(* CODESYS project Function Blocks.export

Project tree, tasks and I/O mapping:
  Function Blocks/
    Actuator/
      function block Actuator [ST]: Close, Open
      function block ActuatotLockAssermbler [ST]: AssembleClosingLockCameraClosed, AssembleClosingLockCameraOpen, AssembleOpenAndUpLock, AssembleOpenvacuumLocked
    DepositeProccess/
      function block absCommonDepositeProcessUnitExplorer [ST]: AddDepositeDevice, AddMaterialRawRateData, AddMaterialShutter, AddQuartzReset, AddQuartzShutter, AddThinknessData, DepositeDeviceCheck, DepositeDeviceStart, DepositeDeviceStop, GetDepositeDevice, GetDepositeDeviceSetting, GetMaterialRawRateData, GetMatertialShutter, GetQuartzReset, GetQuartzShutter, GetThinknessData, InitSelectedPosition, MaterialShutterClose, MaterialShutterOpen, NullPtrCheck, QuartzShutterClose, QuartzShutterOpen, QuartzThinknessReset, _getManipulatingVariable, ActualRawRate, ActualThinkness, DeviceManipulatingVariable, DevicePosition, isMaterialShutterAutoMode, isMaterialShutterRemoteMode, SelectedDevice, SelectedDeviceManipualtedValueFB, SelectedDeviceManipulatingValue, SelectedDeviceSetting
      function block absDepositeUnit [ST]: AddDepositeDevice, AddMaterialShutter, AddQuartzResetCommand, AddQuartzShutter, AddRawRateData, AddThinknessData, CloseMaterialShutter, CloseQuartzShutter, OpenMaterialShutter, OpenQuartzShutter, ResetThinkness, StartDepositeDevice, StopDepositeDevice, DeviceAutoMode, DeviceManipulatingVariable, MaterialShutterAutoMode, MaxManipulatingVariable, MinManipulatingVariable, RawRate, Thinkness
      function block CommonDepositeProcess [ST]: getPreheatTimerTrigger, ProcessStage, _acknowledgment, _calcSP, _error, _getSelectedDevice, _initData, _limitSpeedDeposite, _pidAutoMode, _pidManualMode, _predepositeHeating, _qartzOpen, _qartzSensoreHeating, _quartzOpenedDelay, _resultHandler, _sourceShutterOpen, _startHeater, _startPreheatTimer, _startQuartzHeatingTimer, _startQuartzOpenDelayTimer, _stopDeposite, _stopPreheatTimer, _stopQuartzHeatingTimer, _stopQuartzOpenDelayTimer, _TimerCall, _waitCommand, DepositeSPFromPID, depositeThinknessLimit, Dkoeff, getPreheatLeftTimeSecond, getPreheatTime, getQuartzHeatingLeftTimeSecond, getQuartzHeatingTime, getQuartzOpenDelayLeftTimeSecond, getQuartzOpenDelayTime, Ikoeff, PIDAutoMode, pidAutoModeSP, PIDManualVariable, PIDYMax, PIDYMin, Pkoeff, RawRate, SelectedDevicePosition, _preheatTimerComplete, _quartzHeatingTimerComplete, _quartzOpenDelayTimerComplete
      function block fbDepositeProccess [ST]: AssemblePermition, CalcSP, InitTimers, SelectDepositeSource, Update, getPreheatTimeLeftSecond, setGorn1, setGorn2, setGorn3, setGornSetting1, setGornSetting2, setGornSetting3, setQartzReset1, setQartzReset2, setQartzReset3, setQuartzShutter1, setQuartzShutter2, setQuartzShutter3, setRawRate1, setRawRate2, setRawRate3, setShutter1, setShutter2, setShutter3, setShutterSetting1, setShutterSetting2, setShutterSetting3, setThinkness1, setThinkness2, setThinkness3
      function block fbGornDepositeProccess [ST]: AssemblePermition, CalcSP, InitTimers, SelectDepositeSource, Update, getPreheatTimeLeftSecond, setGorn1, setGorn2, setGorn3, setGornSetting1, setGornSetting2, setGornSetting3, setQartzReset1, setQartzReset2, setQartzReset3, setQuartzShutter1, setQuartzShutter2, setQuartzShutter3, setRawRate1, setRawRate2, setRawRate3, setShutter1, setShutter2, setShutter3, setShutterSetting1, setShutterSetting2, setShutterSetting3, setThinkness1, setThinkness2, setThinkness3
      function block GornDepositeUnit [ST]: _addDepositeDevice, _deviceAutoMode, _deviceManipulatingVariableGet, _deviceManipulatingVariableSet, _maxManipulatingVariable, _minManipulatingVariable, _startDepositeDevice, _stopDepositeDevice
      function block HeaterDepositeUnit [ST]: _addDepositeDevice, _deviceAutoMode, _deviceManipulatingVariableGet, _deviceManipulatingVariableSet, _maxManipulatingVariable, _minManipulatingVariable, _startDepositeDevice, _stopDepositeDevice
    Driver/
      function block fbBSDDriver [ST]
    GasRegulator/
      function block fbGasRegulator [ST]: CalcRRGSPwithCoeff
    GeneralBuffer/
      function block fbGeneralBuffer [ST]: AddElement, AddStruct, ClearBuffer, getBufferAddres, getBufferLength
    Gorn/
      function block Gorn [ST]
    Heater/
      data type udtHeater
      data type udtHeaterSetting
      function block fbHeater [ST]
    Inficon/
      function block fbInficon [ST]: ADD_Sensore, CalcCRC, GetMateriaFiltredRate, HCPub, HelloCommand, RemoteGeneralAction, SensoreStatus
      function block fbInficonQuery [ST]: General, Material, ProcessMaterial, Sensor, Source
      function block fbInficonRemote [ST]: General, MaterialAction
      function block fbInficonStatus [ST]: Material, Sensor
      function block fbInficonUpdate [ST]: General, Material, ProcessMaterial, Sensor, Source
    IPS/
      function block IPSIon [ST]
      function block IPSIonModbus [ST]
    Pumps/
      Interlock/
        function block PumpsInterlock [ST]: AssembleFVPInterlock, AssembleFVPOpenCameraLocked, AssembleTMPFVPTurnOffLocked, AssembleTMPInterlock, AssembleTMPPressureLocked
      function block FVP [ST]: AssebleLock
      function block TMP [ST]: AssembleLock, AssembleLockWithSHV, RotateSignalAssemble, StatusAssemble, StatusTimerLogic
      function block TMPPfifer [ST]
    RRG/
      function block fbRRG [ST]
      function block fbRRGModbus [ST]: AssembleStatusFromFieldStatus2, ConvertModbusSPFeedbackToSPfeedback, ConvertModbusValueFbTovalueFb, ConvertValueSPtoModbusData, UnmarshalModbusFlagStatus1ToRRGFeedback
    Shutter/
      function block fbShutter [ST]
    TRM-151/
      Middleware/
        function block MC_ChannelView_ChannelTRM [ST]
        function block MC_InputView_InputTRM [ST]
        function block MC_OperatingView_OperatingTRM [ST]
        function block MC_OutputView_OutputTRM [ST]
        function block MC_ProgramOfTecholog_ProgramOfTechnologTRM [ST]
        function block MC_RegulatorView_RegulatorTRM [ST]
      Pooling/
        function block MC_TRMPooling [ST]
    TRM_View/
      function block MC_Heater [ST]
      function block MC_TRMChannel [ST]
      function block MC_TRMInput [ST]
      function block MC_TRMOperating [ST]
      function block MC_TRMOutput [ST]
      function block MC_TRMProgramOfTechnolog [ST]
      function block MC_TRMRegulator [ST]
    VacuumCamera/
      Pumping/
        function block VacuumCameraWithoutSHV [ST]: StartDevacuumProcessCommand, StartVacuumProcessCommand, StopVacuumProcessCommand, CancelOperatorCommand, CheckFVPSelect, CheckingFVP, CloseAllvalves, devcuumProcessOpenCam, ErrorHandle, forvacuumingProcess, forvacuumingWithTMPValve, OperatorCommandHandler, operatorStopAnyProcess, startDevacuumProcess, startTMP, startVacuumProcess, stopFVP, stopTMP, stopVacuumProcess, waitVacuumingProcess, isAllValvesClosed, isFVPChecked, isOperatorCommandEntryLocked, isVacuumCameraClosed, isVacuumCameraDeviceAutoMode
        function block VacuumingCameraWithSHV [ST]: CloseAllValves, Devacuum, Revacuum, StartUnit, StopUnit, ValveOpen, _commandHandler, _commandRouter, _resetAllCommand, _resetProcess, isAllvalveClosed
      global variables VacuumCameraErrorsList
      global variables VacuumCameraStatusList
    VacuumSensore/
      ConverExp/
        function ConverPressureToHmi [ST]
        function LessPressure [ST]
        function More [ST]
      function block VacuumSensore [ST]: CalcPressure
    Valves/
      global variables ValveInterlockStatus
      function block Valve [ST]
      function block ValvesInterlock [ST]: AnotherValveOpenInterlock, AssembleSHVLockStatus, AssembleValveStatus, LowPressureInterlock
    function block DiscreteInput [ST]
    function block DiscreteOutput [ST]
    function block HeatFloatSensore [ST]: isFloatL, isFloatLL, isTemepratureHH, isTemperatureH
    function block OwenAnalogInput [ST]
    function block TMPBreakingValve [ST]
*)

// Function Blocks/Heater/udtHeater
TYPE udtHeater :
STRUCT
	xPowerOn:		BOOL;
	xError:			BOOL;
	xLock:			BOOL;
	xManualCommand:	BOOL;
	xAutoCommand:	BOOL;
	xReset:			BOOL;
	xCommand: 		BOOL;
	Temepature:		REAL;
	rPower:			REAL;
	wState:			BYTE;
END_STRUCT
END_TYPE

// Function Blocks/Heater/udtHeaterSetting
TYPE udtHeaterSetting :
STRUCT
	rMinPower:		REAL:=0;
	rMaxPower:		REAL:=100.0;
	rManualPower: 	REAL;
	rAutoPower:		REAL;
	rSetpointTemperature: REAL;
	P: REAL:=2.0;
	I:REAL:=15.0;
	D:REAL:=0.0;
	rMinimalAccessPressure:	REAL:=0.003;
	xAutoMode:		BOOL;
	xServiceMode:	BOOL;
	xManualPower: BOOL;
	
END_STRUCT
END_TYPE

// Function Blocks/VacuumCamera/VacuumCameraErrorsList
{attribute 'qualified_only'}
VAR_GLOBAL CONSTANT
	NO_ERROR: 						WORD:=16#00;
	ALL_DEVICES_DONT_HAVE_AUTOMODE: WORD:=16#02;
	VACUUM_CAMERA_OPEN: 			WORD:=16#03;
	FVP_CHECK_FAIL:					WORD:=16#04;
	TMP_ERROR_FROM_START:			WORD:=16#05;
END_VAR

// Function Blocks/VacuumCamera/VacuumCameraStatusList
{attribute 'qualified_only'}
VAR_GLOBAL CONSTANT
	SYSTEM_READY_AND_WAIT_COMMAND: 			WORD:=00;
	SYSTEM_HAS_ERROR:						WORD:=01;
	STOP_ANY_PROCESS_SIGNAL_FROM_OPERATOR:	WORD:=02;
	START_VACUUM_PROCESS:					WORD:=03;
	CHECK_FVP_START_FVP:					WORD:=04;
	CHECK_FVP_START_TIMER:					WORD:=05;
	CHECK_FVP_COMPLETE:						WORD:=06;
	CHECK_FVP_FAILED:						WORD:=07;
	START_FORVAC_PROCESS:					WORD:=08;
	FORVAC_COMPLETE:						WORD:=09;	
	FORVAC_WITH_TMP_VALVE:					WORD:=10;
	FORVAC_WITH_TMP_VALVE_COMPLETE:			WORD:=11;
	TMP_IS_STARTED:							WORD:=12;
	TMP_IS_RUN:								WORD:=13;
	CAMERA_IS_VACUUMING:					WORD:=14;
	VACUUM_DONE:							WORD:=15;
	STOP_TMP_PROCESS:						WORD:=16;
	STOP_FVP_PROCESS:						WORD:=17;
	STOP_TMP_OPEN_BAV3:						WORD:=18;
	STOP_TMP_DONE:							WORD:=19;
	STOP_FVP_PROCESS_DONE:					WORD:=20;
	STOP_SYSTEM_COMPLITE:					WORD:=21;
	OPERATOR_STOPED_PROCESS_COMPLETE:		WORD:=22;
	BAV3OPENED:								WORD:=23;
	FVP_CHECK_COMPLETED:					WORD:=24;
END_VAR

// Function Blocks/Valves/ValveInterlockStatus
{attribute 'qualified_only'}
VAR_GLOBAL CONSTANT
	NO_LOCK: WORD:=0;//Нет блокировок
	LOW_PRESSURE_INTERLOCK: WORD:=1;//Блокирвока из-за недостаточного давления в пневмосистеме
	LOCKER_VALVE_OPENED: WORD:=2;//Блокировка из-за открытия блокирующего клапана
	HIGH_PRESSURE_INTERLOCK: WORD:=3;// Высокое давление в линии
END_VAR

// Function Blocks/DepositeProccess/absCommonDepositeProcessUnitExplorer/_addDepositeDevice
METHOD PROTECTED ABSTRACT _addDepositeDevice : dpResult
VAR_INPUT
	iPosition: INT;
	ptrDepositeDevice: POINTER TO BYTE;
	ptrDepositeDeviceSetting: POINTER TO BYTE;
END_VAR

// Function Blocks/DepositeProccess/absCommonDepositeProcessUnitExplorer/_addMaterialRawRateData
METHOD PROTECTED ABSTRACT _addMaterialRawRateData : dpResult
VAR_INPUT
	ptrMaterialRawRateData	: POINTER TO BYTE;
	iPosition	: INT;
END_VAR

// Function Blocks/DepositeProccess/absCommonDepositeProcessUnitExplorer/_addMaterialShutter
METHOD PROTECTED ABSTRACT _addMaterialShutter : dpResult
VAR_INPUT
	ptrMaterialShutter	: POINTER TO BYTE;
	ptrMaterialShutterSetting	: POINTER TO BYTE;
	iPosition	: INT;
END_VAR

// Function Blocks/DepositeProccess/absCommonDepositeProcessUnitExplorer/_addQuartzReset
METHOD PROTECTED ABSTRACT _addQuartzReset : dpResult
VAR_INPUT
	ptrQuartzReset	: POINTER TO BYTE;
	iPosition	: INT;
END_VAR

// Function Blocks/DepositeProccess/absCommonDepositeProcessUnitExplorer/_addQuartzShutter
METHOD PROTECTED ABSTRACT _addQuartzShutter : dpResult
VAR_INPUT
	ptrQuartzShutter	: POINTER TO udtDiscreteSignal;
	iPosition	: INT;
END_VAR

// Function Blocks/DepositeProccess/absCommonDepositeProcessUnitExplorer/_addThinknessData
METHOD PROTECTED ABSTRACT _addThinknessData : dpResult
VAR_INPUT
	ptrThinknessData	: POINTER TO REAL;
	iPosition	: INT;
END_VAR

// Function Blocks/DepositeProccess/absCommonDepositeProcessUnitExplorer/_depositeDeviceCheck
METHOD PROTECTED ABSTRACT _depositeDeviceCheck : dpResult
VAR_INPUT
	Status: REFERENCE TO dpuStatus;
END_VAR

// Function Blocks/DepositeProccess/absCommonDepositeProcessUnitExplorer/_depositeDeviceStart
METHOD PROTECTED ABSTRACT _depositeDeviceStart : dpResult
VAR_INPUT
END_VAR

// Function Blocks/DepositeProccess/absCommonDepositeProcessUnitExplorer/_depositeDeviceStop
METHOD PROTECTED ABSTRACT _depositeDeviceStop : dpResult
VAR_INPUT
END_VAR

// Function Blocks/DepositeProccess/absCommonDepositeProcessUnitExplorer/_getDepositeDevice
METHOD PROTECTED ABSTRACT _getDepositeDevice : POINTER TO BYTE
VAR_INPUT
	iPostion	: INT;
END_VAR
VAR_OUTPUT
	Result	: dpResult;
END_VAR

// Function Blocks/DepositeProccess/absCommonDepositeProcessUnitExplorer/_getDepositeDeviceSetting
METHOD PROTECTED ABSTRACT _getDepositeDeviceSetting : POINTER TO BYTE
VAR_INPUT
	iPosition	: INT;
END_VAR
VAR_OUTPUT
	Result	: dpResult;
END_VAR

// Function Blocks/DepositeProccess/absCommonDepositeProcessUnitExplorer/_getMaterialRawRateData
METHOD PROTECTED ABSTRACT _getMaterialRawRateData : POINTER TO REAL
VAR_INPUT
	iPosition	: INT;
END_VAR
VAR_OUTPUT
	Result	: dpResult;
END_VAR

// Function Blocks/DepositeProccess/absCommonDepositeProcessUnitExplorer/_getMaterialShutter
METHOD PROTECTED ABSTRACT _getMaterialShutter : POINTER TO udtShutter
VAR_INPUT
	iPosition	: INT;
END_VAR
VAR_OUTPUT
	Result	: dpResult;
END_VAR

// Function Blocks/DepositeProccess/absCommonDepositeProcessUnitExplorer/_getMaterialShutterSetting
METHOD PROTECTED ABSTRACT _getMaterialShutterSetting : POINTER TO udtShutterSetting
VAR_INPUT
	iPosition	: INT;
END_VAR
VAR_OUTPUT
	Result	: dpResult;
END_VAR

// Function Blocks/DepositeProccess/absCommonDepositeProcessUnitExplorer/_getQuartzReset
METHOD PROTECTED ABSTRACT _getQuartzReset : POINTER TO BOOL
VAR_INPUT
	iPosition	: INT;
END_VAR
VAR_OUTPUT
	Result	: dpResult;
END_VAR

// Function Blocks/DepositeProccess/absCommonDepositeProcessUnitExplorer/_getQuartzShutter
METHOD PROTECTED ABSTRACT _getQuartzShutter : POINTER TO udtDiscreteSignal
VAR_INPUT
	iPosition	: INT;
END_VAR
VAR_OUTPUT
	Result	: dpResult;
END_VAR

// Function Blocks/DepositeProccess/absCommonDepositeProcessUnitExplorer/_getSelectedDepositeDevice
METHOD PROTECTED ABSTRACT _getSelectedDepositeDevice : POINTER TO BYTE
VAR_INPUT
END_VAR

// Function Blocks/DepositeProccess/absCommonDepositeProcessUnitExplorer/_getSelectedDeviceManipulatingValue
{warning 'Проследить за всеми использованиями данного метода'}
METHOD PROTECTED ABSTRACT _getSelectedDeviceManipulatingValue : POINTER TO BYTE
VAR_INPUT
END_VAR

// Function Blocks/DepositeProccess/absCommonDepositeProcessUnitExplorer/_getSelectedDeviceManipulatingValueFB
{warning 'Проследить за всеми использованиями данного метода'}
METHOD PROTECTED ABSTRACT _getSelectedDeviceManipulatingValueFB : POINTER TO BYTE
VAR_INPUT
END_VAR

// Function Blocks/DepositeProccess/absCommonDepositeProcessUnitExplorer/_getSelectedDeviceSetting
METHOD PROTECTED ABSTRACT _getSelectedDeviceSetting : POINTER TO BYTE
VAR_INPUT
END_VAR

// Function Blocks/DepositeProccess/absCommonDepositeProcessUnitExplorer/_getThinknessData
METHOD PROTECTED ABSTRACT _getThinknessData : POINTER TO REAL
VAR_INPUT
	iPosition	: INT;
END_VAR
VAR_OUTPUT
	Result	: dpResult;
END_VAR

// Function Blocks/DepositeProccess/absCommonDepositeProcessUnitExplorer/_initSelectedPosition
//инициализация выбранной позиции. Устройства нагрева
METHOD PROTECTED ABSTRACT _initSelectedPosition : dpResult
VAR_INPUT
	iPosition	: INT;
END_VAR
VAR_OUTPUT
	Status	: dpuStatus;
END_VAR

// Function Blocks/DepositeProccess/absCommonDepositeProcessUnitExplorer/_isDepositeDeviceAutoMode
METHOD PROTECTED ABSTRACT _isDepositeDeviceAutoMode : dpResult
VAR_INPUT
END_VAR

// Function Blocks/DepositeProccess/absCommonDepositeProcessUnitExplorer/_isDepositeDeviceBlocked
METHOD PROTECTED ABSTRACT _isDepositeDeviceBlocked : dpResult
VAR_INPUT
END_VAR

// Function Blocks/DepositeProccess/absCommonDepositeProcessUnitExplorer/_isDepositeDeviceModbusConnected
METHOD PROTECTED ABSTRACT _isDepositeDeviceModbusConnected : dpResult
VAR_INPUT
END_VAR

// Function Blocks/DepositeProccess/absCommonDepositeProcessUnitExplorer/_materialShutterClose
METHOD PROTECTED ABSTRACT _materialShutterClose : dpResult
VAR_INPUT
END_VAR

// Function Blocks/DepositeProccess/absCommonDepositeProcessUnitExplorer/_nullPtrCheck
METHOD PROTECTED ABSTRACT _nullPtrCheck : dpResult
VAR_INPUT
END_VAR

// Function Blocks/DepositeProccess/absCommonDepositeProcessUnitExplorer/_setManipulatingVariable
METHOD PROTECTED ABSTRACT _setManipulatingVariable : dpResult
VAR_INPUT
	Value:REAL;
END_VAR

// Function Blocks/DepositeProccess/absDepositeUnit/_addDepositeDevice
METHOD  ABSTRACT _addDepositeDevice : dpResult
VAR_INPUT
	ptrDevice	: 			POINTER TO BYTE;
	ptrDeviceSetting	: 	POINTER TO BYTE;
END_VAR

// Function Blocks/DepositeProccess/absDepositeUnit/_deviceAutoMode
METHOD PROTECTED ABSTRACT _deviceAutoMode : BOOL
VAR_INPUT
END_VAR

// Function Blocks/DepositeProccess/absDepositeUnit/_deviceManipulatingVariableGet
METHOD PROTECTED ABSTRACT _deviceManipulatingVariableGet : REAL
VAR_INPUT
END_VAR

// Function Blocks/DepositeProccess/absDepositeUnit/_deviceManipulatingVariableSet
METHOD PROTECTED ABSTRACT _deviceManipulatingVariableSet : dpResult
VAR_INPUT
	Variable: REAL;
END_VAR

// Function Blocks/DepositeProccess/absDepositeUnit/_maxManipulatingVariable
METHOD PROTECTED ABSTRACT _maxManipulatingVariable : REAL
VAR_INPUT
END_VAR

// Function Blocks/DepositeProccess/absDepositeUnit/_minManipulatingVariable
METHOD PROTECTED ABSTRACT _minManipulatingVariable : REAL
VAR_INPUT
END_VAR

// Function Blocks/DepositeProccess/absDepositeUnit/_startDepositeDevice
METHOD PROTECTED ABSTRACT _startDepositeDevice : dpResult
VAR_INPUT
	wStatus	: REFERENCE TO dpuStatus;
END_VAR

// Function Blocks/DepositeProccess/absDepositeUnit/_stopDepositeDevice
METHOD PROTECTED ABSTRACT _stopDepositeDevice : dpResult
VAR_INPUT
	wStatus	: REFERENCE TO dpuStatus;
END_VAR

// Function Blocks/DiscreteInput
(*Дискретный входной сигнал*)
FUNCTION_BLOCK DiscreteInput
VAR_INPUT
	Input:						BOOL;//Входной Сигнал
	refDiscreteSignal:			REFERENCE TO udtDiscreteSignal;					//Ссылка на объекта типа "udtDiscreteSignal"
	refDiscreteSignalSetting: 	REFERENCE TO udtDiscreteSignalSetting;			//Настрйоки сигнала
END_VAR
VAR_OUTPUT

END_VAR
VAR
	
END_VAR

refDiscreteSignal.xSignal:=Input;

{region "SimModeService"}
IF NOT refDiscreteSignalSetting.xSimMode THEN
	refDiscreteSignal.xValue:=refDiscreteSignal.xSignal;
ELSE
	refDiscreteSignal.xValue:=refDiscreteSignalSetting.xSimValue;
END_IF
{endregion}
	 
{region "Invertion Service"}
IF refDiscreteSignalSetting.xInv THEN
	refDiscreteSignal.xValue:=NOT refDiscreteSignal.xValue;		 
END_IF
{endregion}

END_FUNCTION_BLOCK

// Function Blocks/DiscreteOutput
(*Дискретный выходной сигнал*)
FUNCTION_BLOCK DiscreteOutput
VAR_INPUT
	refDiscreteSignal: 			REFERENCE TO udtDiscreteSignal;
	refDiscreteSignalSetting:	REFERENCE TO udtDiscreteSignalSetting;
END_VAR
VAR_OUTPUT
	Signal: BOOL;
END_VAR
VAR
END_VAR

{region "Simulation service"}
IF NOT refDiscreteSignalSetting.xSimMode THEN
	refDiscreteSignal.xSignal:=refDiscreteSignal.xValue;
ELSE
	refDiscreteSignal.xSignal:=refDiscreteSignalSetting.xSimValue;
END_IF
{endregion}
	 
{region "Invertion service"}
IF refDiscreteSignalSetting.xInv THEN
	refDiscreteSignal.xSignal:=NOT refDiscreteSignal.xSignal;		 
END_IF
{endregion}


Signal:=refDiscreteSignal.xSignal;

END_FUNCTION_BLOCK

// Function Blocks/HeatFloatSensore
FUNCTION_BLOCK HeatFloatSensore
VAR_INPUT
	refSensore:				REFERENCE TO udtHeatFloatSensore;
	refSensoreSetting:		REFERENCE TO udtHeatFloatSensoreSetting;
	rTemperature:			REAL;
	rFloat:					REAL;
END_VAR
VAR_OUTPUT
	xTemperatureH:			BOOL;
	xTemperatureHH:			BOOL;
	xFloatL:				BOOL;
	xFloatLL:				BOOL;
END_VAR
VAR
END_VAR

refSensore.rInputFloat:=rFloat;
refSensore.rInputTemperature:=rTemperature;

IF refSensore.rInputFloat<0.0 THEN
	refSensore.xErrorFloat:=TRUE;
ELSE
	refSensore.xErrorFloat:=FALSE;
END_IF
IF refSensore.rInputTemperature< -10.0 THEN
	refSensore.xErrorHeat:=TRUE;
ELSE
	refSensore.xErrorHeat:=FALSE;
END_IF

{region "Temeprature"}

	 

	 


{endregion}
{region "Float"}

	 

{endregion}
{region "OUTPUT"}
xTemperatureH:=isTemperatureH;
xTemperatureHH:=isTemepratureHH;
xFloatL:=isFloatL;
xFloatLL:=isFloatLL;
{endregion}

PROPERTY PROTECTED isFloatL : BOOL
GET
IF refSensore.rInputFloat<refSensoreSetting.rFloatSPL AND refSensore.rInputFloat>refSensoreSetting.rFloatSPLL AND NOT refSensore.xFloatLL THEN
	refSensore.xFloatL:=TRUE;
ELSIF refSensore.rInputFloat >refSensoreSetting.rFloatSPL+refSensoreSetting.rFloatHyst THEN
	refSensore.xFloatL:=FALSE;
ELSIF  refSensore.rInputFloat < refSensoreSetting.rFloatSPLL THEN
	refSensore.xFloatL:=FALSE;
END_IF

isFloatL:=refSensore.xFloatL;
END_GET
END_PROPERTY

PROPERTY isFloatLL : BOOL
GET
IF refSensore.rInputFloat < refSensoreSetting.rFloatSPLL THEN
	refSensore.xFloatLL:=TRUE;	
ELSIF refSensore.rInputFloat >refSensoreSetting.rFloatSPLL+refSensoreSetting.rFloatHyst THEN
	refSensore.xFloatLL:=FALSE; 
END_IF
isfloatLL:=refSensore.xFloatLL;
END_GET
END_PROPERTY

PROPERTY PROTECTED isTemepratureHH : BOOL
GET
IF refSensore.rInputTemperature>refSensoreSetting.rTemperatureSPHH  THEN
 	refSensore.xTemperatureHH:=TRUE;	
ELSIF refSensore.rInputTemperature<refSensoreSetting.rTemperatureSPHH-refSensoreSetting.rTemperatureHyst THEN
	refSensore.xTemperatureHH:=FALSE;		 
END_IF		 

isTemepratureHH:=refsensore.xTemperatureHH;
END_GET
END_PROPERTY

PROPERTY PROTECTED isTemperatureH : BOOL
GET
IF refSensore.rInputTemperature>refSensoreSetting.rTemperatureSPH AND refSensore.rInputTemperature<refSensoreSetting.rTemperatureSPHH AND NOT refSensore.xTemperatureHH THEN
 	refSensore.xTemperatureH:=TRUE;	 
ELSIF refSensore.rInputTemperature<refSensoreSetting.rTemperatureSPH-refSensoreSetting.rTemperatureHyst THEN
	refSensore.xTemperatureH:=FALSE;		
ELSIF refSensore.rInputTemperature>refSensoreSetting.rTemperatureSPHH  THEN
 	refSensore.xTemperatureH:=FALSE;			  
END_IF 
	
isTemperatureH:=refSensore.xTemperatureH;
END_GET
END_PROPERTY

END_FUNCTION_BLOCK

// Function Blocks/OwenAnalogInput
FUNCTION_BLOCK OwenAnalogInput
VAR_INPUT
	rSignal:	REAL;
	refAnalogInput:	REFERENCE TO udtOwenAnalogSignal;
END_VAR
VAR_OUTPUT
END_VAR
VAR
END_VAR

refAnalogInput.rSignal:=rSignal;

IF refAnalogInput.xSimMode THEN
	refAnalogInput.rValue:=refAnalogInput.rSimValue;
ELSE
	refAnalogInput.rValue:=refAnalogInput.rSignal;
END_IF

END_FUNCTION_BLOCK

// Function Blocks/TMPBreakingValve
FUNCTION_BLOCK TMPBreakingValve
VAR_INPUT
	TMPBreakinValve: 	REFERENCE TO udtTMPBreakingValve;
	Interlock:			BOOL;
END_VAR
VAR_OUTPUT
	Signal:				BOOL;
END_VAR
VAR
END_VAR

TMPBreakinValve.xInterlock := Interlock;



IF TMPBreakinValve.xAutoMode THEN
	TMPBreakinValve.xManualCommand:=TMPBreakinvalve.xAutoCommand;
	TMPBreakinValve.xOutputCommnad:=TMPBreakinvalve.xAutoCommand;
ELSE
	TMPBreakinValve.xAutoCommand:=TMPBreakinValve.xManualCommand;
	TMPBreakinValve.xOutputCommnad:=TMPBreakinValve.xManualCommand;
END_IF
IF TMPBreakinValve.xInterlock THEN
	TMPBreakinValve.xAutoCommand:=FALSE;
	TMPBreakinValve.xManualCommand:=FALSE;
	TMPBreakinValve.xOutputCommnad:=FALSE;
END_IF

TMPBreakinValve.xOpened:=TMPBreakinValve.xOutputCommnad;
Signal:=TMPBreakinValve.xOutputCommnad;

END_FUNCTION_BLOCK

// Function Blocks/Actuator/Actuator
{attribute 'test'}
FUNCTION_BLOCK Actuator
VAR_INPUT
	refActuator: 		REFERENCE TO udtActuator;
	BAV3:				REFERENCE TO udtValve;
	CameraClosed:		REFERENCE TO udtDiscreteSignal;

	
END_VAR
VAR_OUTPUT
	xOpenSignal:	BOOL;
	xCloseSignal:	BOOL;
END_VAR
VAR
END_VAR

{region "INTERLOCK"}

IF refActuator.xOpenInterlock AND NOT refActuator.xServiceMode THEN
	refActuator.xOpenBlocked:=TRUE;
ELSE
	refActuator.xOpenBlocked:=FALSE;		 
END_IF
IF refActuator.xCloseInterlock AND NOT refActuator.xServiceMode THEN
	refActuator.xCloseBlocked :=TRUE;
ELSE
	refActuator.xCloseBlocked:=FALSE;		 
END_IF
{endregion}

{region "Command Logic"}
Open();
Close();
{endregion}

IF refActuator.xOpen AND CameraClosed.xValue THEN
	BAV3.xAutoCommand:=TRUE;
ELSIF refActuator.xOpen AND NOT CameraClosed.xValue THEN
	BAV3.xAutoCommand:=FALSE;
END_IF

xOpenSignal:=refActuator.xOpen;
xCloseSignal:=refActuator.xClose;

METHOD PROTECTED Close
VAR_INPUT
END_VAR
IF refActuator.xCloseCommand AND NOT refActuator.xCloseBlocked AND NOT refActuator.xOpenCommand THEN
	refActuator.xClose:=TRUE;
ELSE
	refActuator.xClose:=FALSE;
END_IF
END_METHOD

METHOD PROTECTED Open
VAR_INPUT
END_VAR
IF refActuator.xOpenCommand AND NOT refActuator.xOpenBlocked AND NOT refActuator.xCloseCommand THEN
	refActuator.xOpen:=TRUE;
ELSE
	refActuator.xOpen:=FALSE;
END_IF
END_METHOD

END_FUNCTION_BLOCK

// Function Blocks/Actuator/ActuatotLockAssermbler
FUNCTION_BLOCK ActuatotLockAssermbler
VAR_INPUT
	refActuator: 				REFERENCE TO udtActuator;
	CameraPressure:				REFERENCE TO udtPressureSensore;
	CameraPressureMinSetting:	REAL;//Давление ниже которого срабатывает блокировка на открытие
	xCameraVacuumSignal:		BOOL;
	xOpenCameraSignal:			BOOL;
	xUpCameraSignal:			BOOL;
	xClosedCamerSignal:			BOOL;
END_VAR
VAR_OUTPUT
END_VAR
VAR
	xOpenVaccuumLocked:			BOOL; //Блокировка на открытие камеры при вакууме внутри
	xOpenAndUpLock:				BOOL; //Блокировка на открытие камеры при уже открытой камере или при камере в верхнем положении
	xClosingLockCameraOpen:		BOOL; //Блокировка на закрытие камеры если камер открыта
	xClosingLockCameraClosed:	BOOL; //Блокировка на закрытие камеры если камера уже закрыта
END_VAR

xOpenVaccuumLocked:=AssembleOpenvacuumLocked(xCameraVacuumSignal:=THIS^.xCameraVacuumSignal);
xOpenAndUpLock:=AssembleOpenAndUpLock(xOpenCameraSignal:= THIS^.xOpenCameraSignal,
										xUpCameraSignal:= THIS^.xUpCameraSignal);
										
xClosingLockCameraOpen:=AssembleClosingLockCameraOpen(xOpenedCameraSignal:=xOpenCameraSignal);
xClosingLockCameraClosed:=AssembleClosingLockCameraClosed(xClosedCameraSignal:=THIS^.xClosedCamerSignal);


THIS^.refActuator.xOpenInterlock:=xOpenVaccuumLocked OR xOpenAndUpLock;
THIS^.refActuator.xCloseInterlock:=xClosingLockCameraClosed OR xClosingLockCameraOpen;

METHOD PUBLIC AssembleClosingLockCameraClosed : BOOL
VAR_INPUT
	xClosedCameraSignal:	BOOL;
END_VAR
AssembleClosingLockCameraClosed:=xClosedCameraSignal;
END_METHOD

METHOD AssembleClosingLockCameraOpen : BOOL
VAR_INPUT
	xOpenedCameraSignal: BOOL;
END_VAR
AssembleClosingLockCameraOpen:= xOpenedCameraSignal;
END_METHOD

METHOD PUBLIC AssembleOpenAndUpLock : BOOL
VAR_INPUT
	xOpenCameraSignal:	BOOL;
	xUpCameraSignal:	BOOL;	
END_VAR
AssembleOpenAndUpLock:=xOpenCameraSignal OR xUpCameraSignal;
END_METHOD

METHOD PUBLIC AssembleOpenvacuumLocked : BOOL
VAR_INPUT
	xCameraVacuumSignal: BOOL;
END_VAR
IF xCameraVacuumSignal OR CameraPressure.rPressure<THIS^.CameraPressureMinSetting THEN
	AssembleOpenvacuumLocked:=TRUE;
ELSE
	AssembleOpenvacuumLocked:=FALSE;
END_IF
END_METHOD

END_FUNCTION_BLOCK

// Function Blocks/DepositeProccess/absCommonDepositeProcessUnitExplorer
FUNCTION_BLOCK ABSTRACT absCommonDepositeProcessUnitExplorer IMPLEMENTS itfDepositeProcessUnitExplorer
VAR_INPUT
	//Setting: REFERENCE TO udtDepositeProccessSetting;
END_VAR
VAR_OUTPUT
END_VAR
VAR
	_materialShutter: 			POINTER TO udtShutter;
	_materialShutterSetting: 	POINTER TO udtShutterSetting;
	_quartzShutter:				POINTER TO udtDiscreteSignal;
	_quartzReset: 				POINTER TO BOOL;
	_materialRawRate:			POINTER TO REAL;
	_actualThinkness:			POINTER TO REAL;
	_iDevicePosition:			INT;	
END_VAR

(*Добавление указателя на  устройства напыления в список всех устройств*)
METHOD AddDepositeDevice : dpResult 
VAR_INPUT
	ptrDevice	: POINTER TO BYTE;
	ptrDeviceSetting	: POINTER TO BYTE;
	iPosition	: INT;
END_VAR
AddDepositeDevice:= THIS^._addDepositeDevice(	iPosition:=iPosition,
							ptrDepositeDevice:=ptrDevice,
							ptrDepositeDeviceSetting:=ptrDeviceSetting);
END_METHOD

(*Метод добавляет указатель на значение скорости напыления в массив*)
METHOD AddMaterialRawRateData : dpResult (*Status*)
VAR_INPUT
	ptrMaterialRawRateData	: POINTER TO BYTE;
	iPosition	: INT;
END_VAR
AddMaterialRawRateData:=THIS^._addMaterialRawRateData(ptrMaterialRawRateData:=ptrMaterialRawRateData,
						iPosition:=iPosition);
END_METHOD

(*Метод добавляет указатель на пневматическую заслонку для материала*)
METHOD AddMaterialShutter : dpResult
VAR_INPUT
	ptrMaterialShutter	: POINTER TO BYTE;
	ptrMaterialShutterSetting	: POINTER TO BYTE;
	iPosition	: INT;
END_VAR
AddMaterialShutter:=THIS^._addMaterialShutter(ptrMaterialShutter, ptrMaterialShutterSetting, iPosition);
END_METHOD

(*Метод добавляющий указатель на команду сброа показателей кварцевого датчика*)
METHOD AddQuartzReset : dpResult
VAR_INPUT
	ptrQuartzReset	: POINTER TO BOOL;
	iPosition	: INT;
END_VAR
AddQuartzReset:=THIS^._addQuartzReset(ptrQuartzReset, iPosition);
END_METHOD

(*Метод добавляющий указатель на команду открытия залсонки кварцевого датчика в массив*)
METHOD AddQuartzShutter : dpResult
VAR_INPUT
	ptrQuartzShutter	: POINTER TO udtDiscreteSignal;
	iPosition	: INT;
END_VAR
AddQuartzShutter:=THIS^._addQuartzShutter(ptrQuartzShutter,iPosition);
END_METHOD

(*Метод добавляющий указатель на толщину напыления в массив*)
METHOD AddThinknessData : dpResult
VAR_INPUT
	ptrThinknessData	: POINTER TO REAL;
	iPosition	: INT;
END_VAR
AddThinknessData:=THIS^._addThinknessData(ptrThinknessData, iPosition);
END_METHOD

METHOD DepositeDeviceCheck : dpResult
VAR_INPUT
	Status: REFERENCE TO dpuStatus;
END_VAR
DepositeDeviceCheck:=THIS^._depositeDeviceCheck(Status);
END_METHOD

(*Метод отвечающий за запуск устройства напыления*)
METHOD DepositeDeviceStart : dpResult//Возвращает DepositeResult
VAR_OUTPUT
	DeviceStatus	: dpuStatus;
END_VAR
VAR
	_deviceResult: dpResult;
END_VAR
DepositeDeviceStart:=DepositeResult.BUSY;
_deviceResult:=THIS^._depositeDeviceCheck(DeviceStatus);
IF  _deviceResult= DepositeResult.ERROR THEN
	DepositeDeviceStart:=DepositeResult.ERROR;
	RETURN;
ELSIF _deviceResult = DepositeResult.COMPLETE THEN
	DepositeDeviceStart:=THIS^._depositeDeviceStart();
END_IF
END_METHOD

METHOD DepositeDeviceStop : dpResult
VAR_OUTPUT
	DeviceStatus	: dpuStatus;
END_VAR
VAR
	_deviceStatus: dpResult;
END_VAR
DepositeDeviceStop:=DepositeResult.BUSY;
_deviceStatus:=THIS^._depositeDeviceCheck(DeviceStatus);
IF  _deviceStatus = DepositeResult.ERROR THEN
	DepositeDeviceStop:=DepositeResult.ERROR;
	RETURN;
ELSIF _deviceStatus = DepositeResult.COMPLETE THEN
	DepositeDeviceStop:=THIS^._depositeDeviceStop();
END_IF
END_METHOD

(*Метод извлекающий указатель на устройство напыления из массива по указанной позиции*)
METHOD GetDepositeDevice : POINTER TO BYTE
VAR_INPUT
	iPostion	: INT;
END_VAR
VAR_OUTPUT
	Status	: WORD;
END_VAR
GetDepositeDevice:=THIS^._getDepositeDevice(iPostion:=iPostion,
											Result=>Status);
END_METHOD

(*Метод извелкающий указатель на структуру с настройками устройства напыления из массива по указанной позиции*)
METHOD GetDepositeDeviceSetting : POINTER TO BYTE
VAR_INPUT
	iPosition	: INT;
END_VAR
VAR_OUTPUT
	Status	: WORD;
END_VAR
GetDepositeDeviceSetting:=THIS^._getDepositeDeviceSetting(iPosition:=iPosition,
															Result=>Status);
END_METHOD

(*Метод извелкающий указатель на скорость напыления из массива по заданной позиции*)
METHOD GetMaterialRawRateData : POINTER TO REAL
VAR_INPUT
	iPosition	: INT;
END_VAR
VAR_OUTPUT
	Status	: WORD;
END_VAR
GetMaterialRawRateData:=THIS^._getMaterialRawRateData(iPosition:=iPosition,
														Result=>Status);
END_METHOD

(*Метод извлекающий указатель на заслонку материала из массива по заданной позиции*)
METHOD GetMatertialShutter : POINTER TO udtShutter
VAR_INPUT
	iPosition	: INT;
END_VAR
VAR_OUTPUT
	Status	: WORD;
END_VAR
GetMatertialShutter:=_getMaterialShutter(iPosition:=iPosition,
										Result=>Status);
END_METHOD

(*Метод извлекающий указатель на команду сброса кварцевого датчика из массива по заданной позиции*)
METHOD GetQuartzReset : POINTER TO BOOL
VAR_INPUT
	iPosition	: INT;
END_VAR
VAR_OUTPUT
	Result	: dpResult;
END_VAR
GetQuartzReset:=THIS^._getQuartzReset(iPosition:=iPosition,
										Result=>Result);
END_METHOD

(*Метод извлекающий указатель на заслонку кварцевого датчика по заданной позиции*)
METHOD GetQuartzShutter : POINTER TO udtDiscreteSignal
VAR_INPUT
	iPosition	: INT;
END_VAR
VAR_OUTPUT
	Result	: dpResult;
END_VAR
GetQuartzShutter:=THIS^._getQuartzShutter(iPosition:=iPosition,
											Result=>Result);
END_METHOD

(*Метод извлекающий указатель на толщину покрытия из массива по заданной позиции*)
METHOD GetThinknessData : POINTER TO REAL
VAR_INPUT
	iPosition	: INT;
END_VAR
VAR_OUTPUT
	Result	: dpResult;
END_VAR
GetThinknessData:=THIS^._getThinknessData(iPosition:=iPosition,
											Result=>Result);
END_METHOD

METHOD InitSelectedPosition : dpResult
VAR_INPUT
END_VAR
VAR_OUTPUT
	Status	: dpuStatus;
END_VAR
VAR
	Result: dpResult;
END_VAR
THIS^._materialShutter:=THIS^._getMaterialShutter(iPosition:=DevicePosition,
													Result=>Result);
IF Result = DepositeResult.ERROR THEN
	Status:=DepositeProcessStatus.INIT_MATERIAL_SHUTTER_ERROR;
	InitSelectedPosition:=DepositeResult.ERROR;
	RETURN;
END_IF

THIS^._materialShutterSetting:=THIS^._getMaterialShutterSetting(iPosition:=DevicePosition,
													Result=>Result);
IF Result = DepositeResult.ERROR THEN
	Status:=DepositeProcessStatus.INIT_MATERIAL_SHUTTER_SETTING_ERROR;
	InitSelectedPosition:=DepositeResult.ERROR;
	RETURN;
END_IF

THIS^._quartzShutter:=THIS^._getQuartzShutter(iPosition:=DevicePosition,
													Result=>Result);
													
IF Result = DepositeResult.ERROR THEN
	Status:=DepositeProcessStatus.INIT_QUARTZ_SHUTTER_SETTING_ERROR;
	InitSelectedPosition:=DepositeResult.ERROR;
	RETURN;
END_IF

THIS^._quartzReset:=THIS^._getQuartzReset(iPosition:=DevicePosition,
													Result=>Result);
													
IF Result = DepositeResult.ERROR THEN
	Status:=DepositeProcessStatus.INIT_QUARTZ_RESET_SETTING_ERROR;
	InitSelectedPosition:=DepositeResult.ERROR;
	RETURN;
END_IF
	
THIS^._materialRawRate:=THIS^._getMaterialRawRateData(iPosition:=DevicePosition,
													Result=>Result);
													
IF Result = DepositeResult.ERROR THEN
	Status:=DepositeProcessStatus.INIT_MATERIAL_RAW_RATE_ERROR;
	InitSelectedPosition:=DepositeResult.ERROR;
	RETURN;
END_IF
													
THIS^._actualThinkness:=THIS^._getThinknessData(iPosition:=DevicePosition,
												Result=>Result);
												
IF Result = DepositeResult.ERROR THEN
	Status:=DepositeProcessStatus.INIT_THINKNESS_DATA_ERROR;
	InitSelectedPosition:=DepositeResult.ERROR;
	RETURN;
END_IF

												
InitSelectedPosition:=THIS^._initSelectedPosition(iPosition:=DevicePosition,
													Status=>Status);
END_METHOD

(*Метод реализцющий логику закрытия задвижки материала*)
METHOD MaterialShutterClose : WORD
VAR_OUTPUT
	ShutterStatus	: WORD;
END_VAR
MaterialShutterClose:=DepositeResult.BUSY;

IF isMaterialShutterAutoMode <> DepositeDeviceStatus.OK THEN
	MaterialShutterClose:=DepositeResult.ERROR;
	ShutterStatus:=isMaterialShutterAutoMode;
	RETURN;
END_IF
IF isMaterialShutterRemoteMode <> DepositeDeviceStatus.OK THEN
	MaterialShutterClose:=DepositeResult.ERROR;
	ShutterStatus:=isMaterialShutterRemoteMode;
	RETURN;
END_IF
_materialShutter^.AutoCommand:=FALSE;
IF NOT _materialShutter^.ShutterOpened THEN
	MaterialShutterClose:=DepositeResult.COMPLETE;
	RETURN;
END_IF
END_METHOD

(*Метод реализцющий логику открытия задвижки материала*)
METHOD MaterialShutterOpen : dpResult
VAR_OUTPUT
	ShutterStatus	: dpuStatus;
END_VAR
MaterialShutterClose:=DepositeResult.BUSY;

IF isMaterialShutterAutoMode <> DepositeDeviceStatus.OK THEN
	MaterialShutterClose:=DepositeResult.ERROR;
	ShutterStatus:=isMaterialShutterAutoMode;
	RETURN;
END_IF
IF isMaterialShutterRemoteMode <> DepositeDeviceStatus.OK THEN
	MaterialShutterClose:=DepositeResult.ERROR;
	ShutterStatus:=isMaterialShutterRemoteMode;
	RETURN;
END_IF
_materialShutter^.AutoCommand:=TRUE;
IF  _materialShutter^.ShutterOpened THEN
	MaterialShutterClose:=DepositeResult.COMPLETE;
	RETURN;
END_IF
END_METHOD

METHOD NullPtrCheck : WORD
NullPtrCheck:=THIS^._nullPtrCheck();
END_METHOD

METHOD QuartzShutterClose : WORD
QuartzShutterClose:=DepositeResult.BUSY;
THIS^._quartzShutter^.xValue:=FALSE;
QuartzShutterClose:=DepositeResult.COMPLETE;
END_METHOD

METHOD QuartzShutterOpen : WORD
QuartzShutterClose:=DepositeResult.BUSY;
THIS^._quartzShutter^.xValue:=TRUE;
QuartzShutterClose:=DepositeResult.COMPLETE;
END_METHOD

METHOD QuartzThinknessReset : WORD
VAR_INPUT
	Status: REFERENCE TO dpuStatus;
END_VAR
QuartzThinknessReset:=DepositeResult.BUSY;
THIS^._quartzReset^:=TRUE;
Status:=DepositeProcessStatus.QUARTZ_THINKNESS_RESETED;
QuartzThinknessReset:=DepositeResult.COMPLETE;
END_METHOD


METHOD PRIVATE _getManipulatingVariable : REAL
VAR_INPUT
	
END_VAR
END_METHOD

PROPERTY ActualRawRate : REAL
GET
ActualRawRate:=THIS^._materialRawRate^;
END_GET
END_PROPERTY

PROPERTY ActualThinkness : REAL
GET
THIS^.ActualThinkness:=THIS^._actualThinkness^;
END_GET
END_PROPERTY


PROPERTY DeviceManipulatingVariable : REAL
GET
DeviceManipulatingVariable:=THIS^._getManipulatingVariable();
END_GET
SET
THIS^._setManipulatingVariable(DeviceManipulatingVariable);
END_SET
END_PROPERTY

PROPERTY DevicePosition : INT
GET
DevicePosition:=THIS^._iDevicePosition;
END_GET
SET
THIS^._iDevicePosition:=DevicePosition;
END_SET
END_PROPERTY


PROPERTY  isMaterialShutterAutoMode : WORD
GET
IF NOT _materialShutterSetting^.AutoMode THEN
	isMaterialShutterAutoMode:=DepositeDeviceStatus.NOT_AUTO_MODE;
ELSE
	isMaterialShutterAutoMode:=DepositeDeviceStatus.OK;
END_IF
END_GET
END_PROPERTY


PROPERTY  isMaterialShutterRemoteMode : WORD
GET
IF NOT _materialShutterSetting^.RemoteMode THEN
	isMaterialShutterRemoteMode:=DepositeDeviceStatus.NOT_REMOTE_MODE;
ELSE
	isMaterialShutterRemoteMode:=DepositeDeviceStatus.OK;
END_IF
END_GET
END_PROPERTY

PROPERTY SelectedDevice : POINTER TO BYTE
GET
SelectedDevice:=THIS^._getSelectedDepositeDevice();
END_GET
END_PROPERTY

{warning 'Проследить за всеми использованиями данного метода'}
PROPERTY SelectedDeviceManipualtedValueFB : POINTER TO BYTE
GET
SelectedDeviceManipualtedValueFB:=THIS^._getSelectedDeviceManipulatingValueFB();
END_GET
END_PROPERTY

{warning 'Проследить за всеми использованиями данного метода'}
PROPERTY SelectedDeviceManipulatingValue : POINTER TO BYTE
GET
SelectedDeviceManipulatingValue:=THIS^._getSelectedDeviceManipulatingValue();
END_GET
END_PROPERTY

PROPERTY SelectedDeviceSetting : POINTER TO BYTE
GET
SelectedDeviceSetting:=THIS^._getSelectedDeviceSetting();
END_GET
END_PROPERTY

END_FUNCTION_BLOCK

// Function Blocks/DepositeProccess/absDepositeUnit
FUNCTION_BLOCK ABSTRACT absDepositeUnit IMPLEMENTS itfDepositeUnit
VAR_INPUT
END_VAR
VAR_OUTPUT
END_VAR
VAR
	ptrMaterialShutter: 		POINTER TO udtShutter;
	ptrMaterialShutterSetting:	POINTER TO udtShutterSetting;
	ptrQuartzShutter:			POINTER TO udtDiscreteSignal;
	ptrThinkness:				POINTER TO REAL;
	ptrRawRate:					POINTER TO REAL;
	ptrQuartzResetCommand:		POINTER TO BOOL;
END_VAR

METHOD AddDepositeDevice : dpResult
VAR_INPUT
	ptrDevice	: 			POINTER TO BYTE;
	ptrDeviceSetting	: 	POINTER TO BYTE;
END_VAR
_addDepositeDevice(ptrDevice, ptrDeviceSetting);
END_METHOD

METHOD AddMaterialShutter : dpResult
VAR_INPUT
	ptrShutter	: POINTER TO udtShutter;
	ptrShutterSetting	: POINTER TO udtShutterSetting;
END_VAR
AddMaterialShutter:=DepositeResult.BUSY;
THIS^.ptrMaterialShutter:=ptrShutter;
THIS^.ptrMaterialShutterSetting:=ptrShutterSetting;
AddMaterialShutter:=DepositeResult.COMPLETE;
END_METHOD

METHOD AddQuartzResetCommand : dpResult
VAR_INPUT
	Command	: POINTER TO BOOL;
END_VAR
AddQuartzResetCommand:=DepositeResult.BUSY;
THIS^.ptrQuartzResetCommand:=Command;
AddQuartzResetCommand:=DepositeResult.COMPLETE;
END_METHOD


METHOD AddQuartzShutter : dpResult
VAR_INPUT
	ptrQuartzShutter	: POINTER TO udtDiscreteSignal;
END_VAR
AddQuartzShutter:=DepositeResult.BUSY;
THIS^.ptrQuartzShutter:=ptrQuartzShutter;
AddQuartzShutter:=DepositeResult.COMPLETE;
END_METHOD

METHOD AddRawRateData : dpResult
VAR_INPUT
	RawRate	: POINTER TO REAL;
END_VAR
AddRawRateData:=DepositeResult.BUSY;
THIS^.ptrRawRate:=RawRate;
AddRawRateData:=DepositeResult.COMPLETE;
END_METHOD

METHOD AddThinknessData : dpResult
VAR_INPUT
	Thinkness	: POINTER TO REAL;
END_VAR
AddThinknessData:=DepositeResult.BUSY;
THIS^.ptrThinkness:=Thinkness;
AddThinknessData:=DepositeResult.COMPLETE;
END_METHOD

(*Закрытие заслонки материала*)
METHOD CloseMaterialShutter : dpResult
VAR_INPUT
	wStatus	: REFERENCE TO dpuStatus;
END_VAR
CloseMaterialShutter:=DepositeResult.BUSY;
THIS^.ptrMaterialShutter^.AutoCommand:=FALSE;
IF THIS^.ptrMaterialShutter^.ShutterOpened THEN
	wStatus:=DepositeProcessStatus.SRCSHUTTER_CLOSED;
	CloseMaterialShutter:=DepositeResult.COMPLETE;
END_IF
END_METHOD

(*Закрытие заслонки кварцевого датчика*)
METHOD CloseQuartzShutter : dpResult
VAR_INPUT
	wStatus	: REFERENCE TO dpuStatus;
END_VAR
CloseQuartzShutter:=DepositeResult.BUSY;
THIS^.ptrQuartzShutter^.xValue:=FALSE;
wStatus:=DepositeProcessStatus.QCLOSE_CLOSED;
CloseQuartzShutter:=DepositeResult.COMPLETE;
END_METHOD

(*Открытие заслонки материала*)
METHOD OpenMaterialShutter : dpResult
VAR_INPUT
	wStatus	: REFERENCE TO dpuStatus;
END_VAR
OpenMaterialShutter:=DepositeResult.BUSY;
THIS^.ptrMaterialShutter^.AutoCommand:=TRUE;
IF NOT THIS^.ptrMaterialShutter^.ShutterOpened THEN
	wStatus:=DepositeProcessStatus.SRCSHUTTER_OPENED;
	OpenMaterialShutter:=DepositeResult.COMPLETE;
END_IF
END_METHOD

(*Открытие кварцевой заслонки*)
METHOD OpenQuartzShutter : dpResult
VAR_INPUT
	wStatus	: REFERENCE TO dpuStatus;
END_VAR
OpenQuartzShutter:=DepositeResult.BUSY;
THIS^.ptrQuartzShutter^.xValue:=TRUE;
wStatus:=DepositeProcessStatus.QOPEN_OPENED;
OpenQuartzShutter:=DepositeResult.COMPLETE;
END_METHOD

(*Сброс толщины*)
METHOD ResetThinkness : dpResult
VAR_INPUT
	wStatus	: REFERENCE TO dpuStatus;
END_VAR
ResetThinkness:=DepositeResult.BUSY;
THIS^.ptrQuartzResetCommand^:=TRUE;
wStatus:=DepositeProcessStatus.QUARTZ_THINKNESS_RESETED;
ResetThinkness:=DepositeResult.COMPLETE;
END_METHOD

(*Запуск напыления*)
METHOD StartDepositeDevice : dpResult
VAR_INPUT
	wStatus	: REFERENCE TO dpuStatus;
END_VAR
StartDepositeDevice:=_startDepositeDevice(wStatus);
END_METHOD

(*Остановка напыления*)
METHOD StopDepositeDevice : dpResult
VAR_INPUT
	wStatus	: REFERENCE TO dpuStatus;
END_VAR
StopDepositeDevice:=THIS^._stopDepositeDevice(wStatus);
END_METHOD

PROPERTY DeviceAutoMode : BOOL
GET
DeviceAutoMode:=THIS^._deviceAutoMode();
END_GET
END_PROPERTY

(*Уставка для управления нагревателя*)
PROPERTY DeviceManipulatingVariable : REAL
GET
DeviceManipulatingVariable:=THIS^._deviceManipulatingVariableGet();
END_GET
SET
THIS^._deviceManipulatingVariableSet(DeviceManipulatingVariable);
END_SET
END_PROPERTY

PROPERTY MaterialShutterAutoMode : BOOL
GET
MaterialShutterAutoMode:=THIS^.ptrMaterialShutterSetting^.AutoMode;
END_GET
END_PROPERTY

PROPERTY MaxManipulatingVariable : REAL
GET
MaxManipulatingVariable:=THIS^._maxManipulatingVariable();
END_GET
END_PROPERTY

PROPERTY MinManipulatingVariable : REAL
GET
MinManipulatingVariable:=THIS^._minManipulatingVariable();
END_GET
END_PROPERTY


PROPERTY RawRate : REAL
GET
RawRate:=THIS^.ptrRawRate^;
END_GET
END_PROPERTY


PROPERTY Thinkness : REAL
GET
Thinkness:=THIS^.ptrThinkness^;
END_GET
END_PROPERTY

END_FUNCTION_BLOCK

// Function Blocks/DepositeProccess/CommonDepositeProcess
FUNCTION_BLOCK CommonDepositeProcess
VAR_INPUT
	
	iDepositeUnitArraySize:		INT;
	
	refDepositeProcessData: 	REFERENCE TO udtDepositeProcessData;
	refDepositeProcessSetting: 	REFERENCE TO udtGornDepositeProccessSetting;
END_VAR
VAR_IN_OUT
	itfDepositeUnitArray: ARRAY[0..4] OF itfDepositeUnit;
END_VAR
VAR_OUTPUT
	Status: dpuStatus;
	Stage: INT;
END_VAR
VAR
	{#region "Timer}
	_preHeatTimer:				TON;//Время препрогрева
	_quartzOpenDelayTimer:		TON;//Время открытия кварцевого датчика до напыления
	_quartzHeatingTimer:		TON;//Время прогрева кварцевого датчика
	
	_preheatLeftTime:			TIME;//(мс)Прошедшее время с момента препрогрева
	_quartzOpenDelayLeftTime:	TIME;//(мс)Прошедшее время с момента открытия кварцевого датчика до наплынеия
	_quartzHeatingLeftTime:		TIME;//(мс)Прошедшее время с момента начала прогрева кварцевого датчика
	
	xPreheatTimerTrigger:		BOOL;
	xQuartzOpenDelayTrigger:	BOOL;
	xQuartzHeatingTrigger:		BOOL;
	{endregion}
	_selectedDepositeDevice: itfDepositeUnit;		 
	_iStage: 		INT;
	_wResult: 		dpResult;
	_wStatus:		dpuStatus;
	_wProcessStatus:WORD;
	xInit: BOOL;
END_VAR

THIS^._TimerCall();

IF refDepositeProcessData.xStopCommand THEN
	refDepositeProcessData.xStopCommand:=FALSE;
	_iStage:=DepositeProcessStage.STOP_DEPOSITE;
END_IF


CASE _iStage OF
	DepositeProcessStage.WAIT_COMMAND:
	IF NOT xInit THEN
		
		_wResult:=THIS^._initData(_wStatus);
		IF _wResult = DepositeResult.COMPLETE THEN
			xInit:=TRUE;
		END_IF
		IF _wResult = DepositeResult.ERROR THEN
			_iStage:=DepositeProcessStage.ERROR;
			RETURN;
		END_IF
	END_IF
	IF xInit THEN
		_iStage:=THIS^._waitCommand(_wStatus,DepositeProcessStage.INIT_DATA);
	END_IF
		
	DepositeProcessStage.INIT_DATA:
		refDepositeProcessData.xStartCommand:=FALSE;
		_wResult:=THIS^._initData(_wStatus);
		_iStage:=THIS^._resultHandler(	wResult:= _wResult,
										wStatus:= _wStatus ,
										CompleteStatus:=DepositeProcessStatus.INIT_DONE,										
										CompleteStage:=DepositeProcessStage.START_HEATER,
										ErrorStage:= DepositeProcessStage.ERROR,
										ActualStage:=DepositeProcessStage.INIT_DATA);
	
	DepositeProcessStage.START_HEATER:
		_wResult:=THIS^._startHeater(_wStatus);
		_iStage:=THIS^._resultHandler(	wResult:= _wResult,
										wStatus:= _wStatus ,
										CompleteStatus:=DepositeProcessStatus.STARTED_HEATER,										
										CompleteStage:=DepositeProcessStage.PREDEPOSITE_HEATING,
										ErrorStage:= DepositeProcessStage.ERROR,
										ActualStage:=DepositeProcessStage.START_HEATER);
										
	DepositeProcessStage.PREDEPOSITE_HEATING:
		_wResult:=THIS^._predepositeHeating(_wStatus);
		_iStage:=THIS^._resultHandler(	wResult:= _wResult,
										wStatus:= _wStatus ,
										CompleteStatus:=DepositeProcessStatus.PREHEAT_PROCESS_COMPLETE,										
										CompleteStage:=DepositeProcessStage.QARTZ_OPEN,
										ErrorStage:= DepositeProcessStage.ERROR,
										ActualStage:=DepositeProcessStage.PREDEPOSITE_HEATING);
		
	DepositeProcessStage.QARTZ_OPEN:
		_wResult:=THIS^._qartzOpen(_wStatus);
		_iStage:=THIS^._resultHandler(	wResult:= _wResult,
										wStatus:= _wStatus ,
										CompleteStatus:=DepositeProcessStatus.QOPEN_OPENED,										
										CompleteStage:=DepositeProcessStage.QUARTZ_OPENED_DELAY,
										ErrorStage:= DepositeProcessStage.ERROR,
										ActualStage:=DepositeProcessStage.QARTZ_OPEN);
	
	DepositeProcessStage.QUARTZ_OPENED_DELAY:
		_wResult:=THIS^._quartzOpenedDelay(_wStatus);
		_iStage:=THIS^._resultHandler(	wResult:= _wResult,
										wStatus:= _wStatus ,
										CompleteStatus:=DepositeProcessStatus.QOPEN_DELAY_COMPLETE,										
										CompleteStage:=DepositeProcessStage.SOURCE_SHUTTER_OPEN,
										ErrorStage:= DepositeProcessStage.ERROR,
										ActualStage:=DepositeProcessStage.QUARTZ_OPENED_DELAY);
	
	DepositeProcessStage.SOURCE_SHUTTER_OPEN:
		_wResult:=THIS^._sourceShutterOpen(_wStatus);
		_iStage:=THIS^._resultHandler(	wResult:= _wResult,
										wStatus:= _wStatus ,
										CompleteStatus:=DepositeProcessStatus.SRCSHUTTER_OPENED,										
										CompleteStage:=DepositeProcessStage.QARTZ_SENSORE_HEATING,
										ErrorStage:= DepositeProcessStage.ERROR,
										ActualStage:=DepositeProcessStage.SOURCE_SHUTTER_OPEN);
										
	DepositeProcessStage.QARTZ_SENSORE_HEATING:
		_wResult:=THIS^._qartzSensoreHeating(_wStatus);
		_iStage:=THIS^._resultHandler(	wResult:= _wResult,
										wStatus:= _wStatus ,
										CompleteStatus:=DepositeProcessStatus.QUARTZ_HEATING_COMPLETE,										
										CompleteStage:=DepositeProcessStage.LIMIT_SPEED_DEPOSITE_1,
										ErrorStage:= DepositeProcessStage.ERROR,
										ActualStage:=DepositeProcessStage.QARTZ_SENSORE_HEATING);
	DepositeProcessStage.LIMIT_SPEED_DEPOSITE_1:
		_wResult:=THIS^._limitSpeedDeposite(wStatus:=_wStatus,
											StartProcessStatus:=DepositeProcessStatus.LIM_SPEEDDEPOSITE_1_START,
											rPIDAutoModeSP:=THIS^.refDepositeProcessSetting.DepositeSpeedSP_2,
											NewThinknessLimit:=THIS^.refDepositeProcessSetting.DepositeThinkness_2);
		_iStage:=THIS^._resultHandler(	wResult:= _wResult,
										wStatus:= _wStatus ,
										CompleteStatus:=DepositeProcessStatus.LIM_SPEEDDEPOSITE_1_COMPLETE,										
										CompleteStage:=DepositeProcessStage.LIMIT_SPEED_DEPOSITE_2,
										ErrorStage:= DepositeProcessStage.ERROR,
										ActualStage:=DepositeProcessStage.LIMIT_SPEED_DEPOSITE_1);
	
	DepositeProcessStage.LIMIT_SPEED_DEPOSITE_2:
				_wResult:=THIS^._limitSpeedDeposite(wStatus:=_wStatus,
											StartProcessStatus:=DepositeProcessStatus.LIM_SPEEDDEPOSITE_2_START,
											rPIDAutoModeSP:=THIS^.refDepositeProcessSetting.DepositeSpeedSP_2,
											NewThinknessLimit:=THIS^.refDepositeProcessSetting.DepositeThinkness_2);
		_iStage:=THIS^._resultHandler(	wResult:= _wResult,
										wStatus:= _wStatus ,
										CompleteStatus:=DepositeProcessStatus.LIM_SPEEDDEPOSITE_2_COMPLETE,										
										CompleteStage:=DepositeProcessStage.STOP_DEPOSITE,
										ErrorStage:= DepositeProcessStage.ERROR,
										ActualStage:=DepositeProcessStage.LIMIT_SPEED_DEPOSITE_2);
	
	DepositeProcessStage.STOP_DEPOSITE:
		_wResult:=THIS^._stopDeposite(THIS^._wStatus);
		_iStage:=THIS^._resultHandler(	wResult:= _wResult,
										wStatus:= _wStatus ,
										CompleteStatus:=DepositeProcessStatus.PROCESS_COMPLETE,										
										CompleteStage:=DepositeProcessStage.WAIT_COMMAND,
										ErrorStage:= DepositeProcessStage.ERROR,
										ActualStage:=DepositeProcessStage.STOP_DEPOSITE);
	
	DepositeProcessStage.ERROR:
		_wResult:=THIS^._error(THIS^._wStatus);
		IF refDepositeProcessData.xAcknowledgment THEN
			refDepositeProcessData.xAcknowledgment:=FALSE;
			_iStage:=THIS^._acknowledgment(DepositeProcessStage.WAIT_COMMAND);
		END_IF
		
END_CASE
Status:=_wStatus;
Stage:=_iStage;

PROPERTY PUBLIC getPreheatTimerTrigger : BOOL
GET
getPreheatTimerTrigger:=THIS^.xPreheatTimerTrigger;
END_GET
END_PROPERTY


PROPERTY PUBLIC ProcessStage : INT
SET
{IF defined (TEST)}
THIS^._iStage:=ProcessStage;
{END_IF}
END_SET
END_PROPERTY

METHOD PROTECTED _acknowledgment : INT
VAR_INPUT
	CompleteStage: INT;
END_VAR
_acknowledgment:=CompleteStage;
END_METHOD

METHOD PROTECTED _calcSP : INT
VAR_INPUT
END_VAR
_calcSP:=(((refDepositeProcessSetting.FinallyPreheatSP-refDepositeProcessSetting.StartPreheatSP)/refDepositeProcessSetting.PreheatingTime)*getPreheatLeftTimeSecond)+refDepositeProcessSetting.StartPreheatSP;
END_METHOD

METHOD PROTECTED _error : dpResult
VAR_INPUT
	wStatus:REFERENCE TO dpuStatus;
END_VAR
END_METHOD

METHOD PROTECTED _getSelectedDevice : dpResult
VAR_INPUT
END_VAR
VAR
	
END_VAR
_getSelectedDevice:=DepositeResult.BUSY;
IF THIS^.SelectedDevicePosition > THIS^.iDepositeUnitArraySize-1 THEN
	_getSelectedDevice:=DepositeResult.ERROR;
	RETURN;
END_IF
THIS^._selectedDepositeDevice:=THIS^.itfDepositeUnitArray[THIS^.SelectedDevicePosition];
{warning 'Реализовать проверку'}
_getSelectedDevice:=DepositeResult.COMPLETE;
END_METHOD

METHOD PROTECTED _initData : dpResult
VAR_INPUT
	wStatus:REFERENCE TO dpuStatus;
END_VAR
VAR
	Result: dpResult;
END_VAR
_initData:=DepositeResult.BUSY;
wStatus:=DepositeProcessStatus.INIT_START;
Result:=THIS^._getSelectedDevice();
IF Result = DepositeResult.ERROR THEN
	_initData := DepositeResult.ERROR;
	RETURN;
END_IF
IF Result=DepositeResult.COMPLETE THEN
	_initData:=DepositeResult.COMPLETE;
END_IF
END_METHOD

METHOD PROTECTED _limitSpeedDeposite : dpResult
VAR_INPUT
	wStatus: REFERENCE TO dpuStatus;
	StartProcessStatus: dpuStatus;
	rPIDAutoModeSP: REAL;
	NewThinknessLimit: REAL;
END_VAR
_limitSpeedDeposite:=DepositeResult.BUSY;
wStatus:=StartProcessStatus;
THIS^._selectedDepositeDevice.DeviceManipulatingVariable:=THIS^.refDepositeProcessData.ManipulatingVariableFromPID;
IF THIS^._selectedDepositeDevice.Thinkness >=depositeThinknessLimit THEN
	_limitSpeedDeposite:=DepositeResult.COMPLETE;
	pidAutoModeSP:=rPIDAutoModeSP;
	depositeThinknessLimit:=NewThinknessLimit;
END_IF
END_METHOD

METHOD PROTECTED _pidAutoMode : dpResult
VAR_INPUT
END_VAR
THIS^.refDepositeProcessData.xPIDManualMode:=FALSE;
END_METHOD

METHOD PROTECTED _pidManualMode : dpResult
VAR_INPUT
END_VAR
THIS^.refDepositeProcessData.xPIDManualMode := TRUE;
END_METHOD

METHOD PROTECTED _predepositeHeating : dpResult;
VAR_INPUT
	wStatus: REFERENCE TO dpuStatus;
END_VAR
VAR
	CalcManipulatedValue: INT;
END_VAR
_predepositeHeating:=DepositeResult.BUSY;
wStatus:=DepositeProcessStatus.PREHEAT_PROCESS_START;
THIS^.refDepositeProcessData.ManualVariableSPtoPID:=THIS^._calcSP();
DepositeSPFromPID:=THIS^.refDepositeProcessData.ManualVariableSPtoPID;
IF _preheatTimerComplete THEN
	wStatus:=DepositeProcessStatus.PREHEAT_PROCESS_COMPLETE;
	_predepositeHeating:=DepositeResult.COMPLETE;
	THIS^._stopPreheatTimer();
END_IF
END_METHOD

METHOD PROTECTED _qartzOpen : dpResult
VAR_INPUT
	wStatus: REFERENCE TO dpuStatus;	
END_VAR
VAR
	Result: dpResult;
END_VAR
_qartzOpen:=DepositeResult.BUSY;
Result:=THIS^._selectedDepositeDevice.OpenQuartzShutter(wStatus);
IF Result = DepositeResult.COMPLETE THEN
	wStatus:=DepositeProcessStatus.QOPEN_OPENED;
	_qartzOpen:=DepositeResult.COMPLETE;
	_startQuartzOpenDelayTimer();
END_IF
END_METHOD

METHOD PROTECTED _qartzSensoreHeating : dpResult
VAR_INPUT
	wStatus: REFERENCE TO dpuStatus;
END_VAR
VAR
	Result: dpResult;
END_VAR
_qartzSensoreHeating:=DepositeResult.BUSY;
IF _quartzHeatingTimerComplete THEN
	THIS^._stopQuartzHeatingTimer();
	Result:=THIS^._selectedDepositeDevice.ResetThinkness(wStatus);
	_qartzSensoreHeating:=DepositeResult.COMPLETE;
	THIS^._pidAutoMode();
	pidAutoModeSP:=THIS^.refDepositeProcessSetting.DepositeSpeedSP_1;
	depositeThinknessLimit:=THIS^.refDepositeProcessSetting.DepositeThinkness_1;
END_IF
END_METHOD

METHOD PROTECTED _quartzOpenedDelay : dpResult
VAR_INPUT
	wStatus: REFERENCE TO dpuStatus;
END_VAR
_quartzOpenedDelay:=DepositeResult.BUSY;
wStatus:=DepositeProcessStatus.QOPEN_DELAY;
IF _quartzOpenDelayTimerComplete THEN
	THIS^._stopQuartzOpenDelayTimer();
	_quartzOpenedDelay:=DepositeResult.COMPLETE;
END_IF
END_METHOD

METHOD PROTECTED _resultHandler : INT
VAR_INPUT
	wResult: REFERENCE TO WORD;
	wStatus: REFERENCE TO WORD;
	CompleteStatus: WORD;
	CompleteStage: INT;
	ErrorStage: INT;
	ActualStage:int;
END_VAR
IF wResult = DepositeResult.COMPLETE THEN
	_resultHandler:=CompleteStage;
	RETURN;
ELSIF _wResult = DepositeResult.ERROR THEN
	_resultHandler:=ErrorStage;
	RETURN;
END_IF
_resultHandler:=ActualStage;
END_METHOD

METHOD PROTECTED _sourceShutterOpen : dpResult
VAR_INPUT
	wStatus: REFERENCE TO dpuStatus;
END_VAR
VAR
	Result: dpResult;
END_VAR
_sourceShutterOpen:=DepositeResult.BUSY;
Result:=THIS^._selectedDepositeDevice.OpenMaterialShutter(wStatus);
IF Result = DepositeResult.ERROR THEN
	_sourceShutterOpen:=DepositeResult.ERROR;
	RETURN;
END_IF
IF Result = DepositeResult.COMPLETE THEN
	THIS^._startQuartzHeatingTimer();
	_sourceShutterOpen := DepositeResult.COMPLETE;
	RETURN;
END_IF
END_METHOD

METHOD PROTECTED _startHeater : dpResult
VAR_INPUT
	wStatus: REFERENCE TO dpuStatus;
END_VAR
VAR
	DepositeDeviceStartResult: dpResult;
END_VAR
_startHeater:=DepositeResult.BUSY;
wStatus:=DepositeProcessStatus.STARTING_HEATER;
THIS^._pidManualMode();
THIS^.refDepositeProcessData.ManualVariableSPtoPID:=THIS^.refDepositeProcessSetting.StartPreheatSP;
DepositeDeviceStartResult:=THIS^._selectedDepositeDevice.StartDepositeDevice(wStatus);
IF DepositeDeviceStartResult = DepositeResult.ERROR THEN
	_startHeater:=DepositeResult.ERROR;
	RETURN;
END_IF
IF DepositeDeviceStartResult = DepositeResult.COMPLETE THEN
	THIS^._startPreheatTimer();
	_startHeater:=DepositeResult.COMPLETE;
	RETURN;
END_IF
END_METHOD

METHOD PROTECTED _startPreheatTimer
VAR_INPUT
END_VAR
THIS^.xPreheatTimerTrigger:=TRUE;
END_METHOD

METHOD PROTECTED _startQuartzHeatingTimer
VAR_INPUT
END_VAR
THIS^.xQuartzHeatingTrigger:=TRUE;
END_METHOD

METHOD PROTECTED _startQuartzOpenDelayTimer
VAR_INPUT
END_VAR
THIS^.xQuartzOpenDelayTrigger:=TRUE;
END_METHOD

METHOD PROTECTED _stopDeposite : dpResult
VAR_INPUT
	wStatus: REFERENCE TO dpuStatus;
END_VAR
VAR
	Result:dpResult;
END_VAR
_stopDeposite:=DepositeResult.BUSY;
Result:=THIS^._selectedDepositeDevice.StopDepositeDevice(wStatus);
IF Result = DepositeResult.ERROR THEN
	_stopDeposite:=DepositeResult.ERROR;
	RETURN;
END_IF
THIS^._pidManualMode();
THIS^.refDepositeProcessData.ManualVariableSPtoPID:=THIS^.refDepositeProcessSetting.FinallyPreheatSP;
THIS^._selectedDepositeDevice.DeviceManipulatingVariable:=THIS^.refDepositeProcessSetting.FinallyPreheatSP;
THIS^._selectedDepositeDevice.CloseMaterialShutter(wStatus:=wStatus);

_stopDeposite:=DepositeResult.COMPLETE;
END_METHOD

METHOD PROTECTED _stopPreheatTimer
VAR_INPUT
END_VAR
THIS^.xPreheatTimerTrigger:=FALSE;
END_METHOD

METHOD PROTECTED _stopQuartzHeatingTimer
VAR_INPUT
END_VAR
THIS^.xQuartzHeatingTrigger:=FALSE;
END_METHOD

METHOD PROTECTED _stopQuartzOpenDelayTimer
VAR_INPUT
END_VAR
THIS^.xQuartzOpenDelayTrigger:=FALSE;
END_METHOD

METHOD PROTECTED _TimerCall
VAR_INPUT
END_VAR
THIS^._preHeatTimer(IN:=xPreheatTimerTrigger,
					PT:=getPreheatTime,
					ET=>THIS^._preheatLeftTime);
					
THIS^._quartzOpenDelayTimer(IN:=xQuartzOpenDelayTrigger,
							PT:=getQuartzOpenDelayTime,
							ET=>THIS^._quartzOpenDelayLeftTime);

THIS^._quartzHeatingTimer(IN:=xQuartzHeatingTrigger,
							PT:=getQuartzHeatingTime,
							ET=>THIS^._quartzHeatingLeftTime);
END_METHOD

METHOD PROTECTED _waitCommand : INT;
VAR_INPUT
	wStatus:REFERENCE TO dpuStatus;
	iStartStage: INT;
END_VAR
wStatus:=DepositeProcessStatus.WAIT_COMMAND;
IF THIS^.refDepositeProcessData.xStartCommand THEN
	_waitCommand:=iStartStage;
	RETURN;
END_IF
END_METHOD

PROPERTY PUBLIC DepositeSPFromPID : REAL
SET
THIS^._selectedDepositeDevice.DeviceManipulatingVariable:=DepositeSPFromPID;
END_SET
END_PROPERTY

PROPERTY depositeThinknessLimit : REAL
GET
depositeThinknessLimit:=THIS^.refDepositeProcessData.rDepositeThinknessLimit;
END_GET
SET
THIS^.refDepositeProcessData.rDepositeThinknessLimit:=depositeThinknessLimit;
END_SET
END_PROPERTY

PROPERTY PUBLIC Dkoeff : REAL
GET
Dkoeff:=THIS^.refDepositeProcessSetting.KD;
END_GET
END_PROPERTY

PROPERTY PUBLIC getPreheatLeftTimeSecond : UINT
GET
getPreheatLeftTimeSecond:=DWORD_TO_UINT(TIME_TO_DWORD(THIS^._preheatLeftTime)/1000);
END_GET
END_PROPERTY

PROPERTY PUBLIC getPreheatTime : TIME
GET
getPreheatTime:=DWORD_TO_TIME(UINT_TO_DWORD(THIS^.refDepositeProcessSetting.PreheatingTime*1000));
END_GET
END_PROPERTY

PROPERTY PUBLIC getQuartzHeatingLeftTimeSecond : UINT
GET
getQuartzHeatingLeftTimeSecond:=TIME_TO_UINT(THIS^._quartzHeatingLeftTime)/1000;
END_GET
END_PROPERTY

PROPERTY PUBLIC getQuartzHeatingTime : TIME
GET
getQuartzHeatingTime:=DWORD_TO_TIME(UINT_TO_DWORD(THIS^.refDepositeProcessSetting.QuartzHeatingTime*1000));
END_GET
END_PROPERTY

PROPERTY PUBLIC getQuartzOpenDelayLeftTimeSecond : UINT
GET
getQuartzOpenDelayLeftTimeSecond:=TIME_TO_UINT(THIS^._quartzOpenDelayLeftTime)/1000;
END_GET
END_PROPERTY

PROPERTY PUBLIC getQuartzOpenDelayTime : TIME
GET
getQuartzOpenDelayTime:=DWORD_TO_TIME(UINT_TO_DWORD(THIS^.refDepositeProcessSetting.QuartzDelayTime*1000));
END_GET
END_PROPERTY

PROPERTY PUBLIC Ikoeff : REAL
GET
Ikoeff:=THIS^.refDepositeProcessSetting.KI;
END_GET
END_PROPERTY

PROPERTY PUBLIC PIDAutoMode : BOOL
GET
PIDAutoMode:=THIS^.refDepositeProcessData.xPIDManualMode;
END_GET
END_PROPERTY

(*Уставка для пид регулятора в автоматическом режиме*)
PROPERTY PUBLIC pidAutoModeSP : REAL
GET
pidAutoModeSP:=THIS^.refDepositeProcessData.rPIDAutoVariableSP;
END_GET
SET
THIS^.refDepositeProcessData.rPIDAutoVariableSP:=pidAutoModeSP;
END_SET
END_PROPERTY

PROPERTY PIDManualVariable : REAL
GET
PIDManualVariable:=THIS^.refDepositeProcessData.ManualVariableSPtoPID;
END_GET
END_PROPERTY

PROPERTY PUBLIC PIDYMax : REAL
GET
PIDYMax:=THIS^._selectedDepositeDevice.MaxManipulatingVariable;
END_GET
END_PROPERTY

PROPERTY PUBLIC PIDYMin : REAL
GET
PIDYMin:=THIS^._selectedDepositeDevice.MinManipulatingVariable;
END_GET
END_PROPERTY

PROPERTY PUBLIC Pkoeff : REAL
GET
Pkoeff:=THIS^.refDepositeProcessSetting.KP;
END_GET
END_PROPERTY

PROPERTY PUBLIC RawRate : REAL
GET
RawRate:=THIS^._selectedDepositeDevice.RawRate;
END_GET
END_PROPERTY

PROPERTY SelectedDevicePosition : INT
GET
SelectedDevicePosition:=THIS^.refDepositeProcessData.iSelectedDevice;
END_GET
END_PROPERTY

PROPERTY PROTECTED _preheatTimerComplete : BOOL
GET
_preheatTimerComplete:=THIS^._preHeatTimer.Q;
END_GET
END_PROPERTY

PROPERTY PROTECTED _quartzHeatingTimerComplete : BOOL
GET
_quartzHeatingTimerComplete:=THIS^._quartzHeatingTimer.Q;
END_GET
END_PROPERTY

PROPERTY PROTECTED _quartzOpenDelayTimerComplete : BOOL
GET
_quartzOpenDelayTimerComplete:=THIS^._quartzOpenDelayTimer.Q;
END_GET
END_PROPERTY

END_FUNCTION_BLOCK

// Function Blocks/DepositeProccess/fbDepositeProccess
FUNCTION_BLOCK fbDepositeProccess
VAR_INPUT
	refStarProcess:				REFERENCE TO BOOL; //Команда на старт процесса
	refAcknowledgment:			REFERENCE TO BOOL; //команда на сброс ошибки.
	refProcessSetting: 			REFERENCE TO udtGornDepositeProccessSetting;
	refProcessData:	   			REFERENCE TO udtGornDepositeProccessData;
END_VAR
VAR_OUTPUT
	Status :					WORD;
END_VAR
VAR
	ptrGornList: 				ARRAY[0..2] OF POINTER TO udtGorn;
	ptrGornSettingList:			ARRAY[0..2] OF POINTER TO udtGornSetting;
	ptrShutterList:				ARRAY[0..2] OF POINTER TO udtShutter;
	ptrShutterSettingList:		ARRAY[0..2] OF POINTER TO udtShutterSetting;
	ptrQuartzShutterList:		ARRAY[0..2] OF POINTER TO udtDiscreteSignal;
	ptrQuartzResetList:			ARRAY[0..2] OF POINTER TO BOOL;
	ptrThinknessList:			ARRAY[0..2] OF POINTER TO REAL;
	ptrMaterialRawRateList:		ARRAY[0..2] OF POINTER TO REAL;
	_ptrGorn:					POINTER TO udtGorn;
	_ptrGornSetting:			POINTER TO udtGornSetting;
	_ptrShutter:				POINTER TO udtShutter;
	_ptrShutterSetting:			POINTER TO udtShutterSetting;
	_ptrQuartzShutter:			POINTER TO udtDiscreteSignal;
	_ptrQuartzReset:			POINTER TO BOOL;
	_ptrThinkness:				POINTER TO REAL;
	_ptrQuartzRawRate:			POINTER TO REAL;
	_preHeatTimer:				TON;//Время препрогрева
	_preheatLeftTime:			TIME;//(мс)Прошедшее время с момента препрогрева
	
	_qartzOpenDelayTimer:		TON;//Время открытия кварцевого датчика до напыления
	_qartzHeatingTimer:			TON;//Время прогрева кварцевого датчика
	_assemblePermitionStatus:	WORD;
	_stage:						INT; //Стадии работы
	
	_permition:					BOOL;//Разрешение на старт процесса
	_selectedGornPermition: 	BOOL;//Разрешение на старт выбранного источника тока
	_selectedShutterPermition:	BOOL;//Разрешение от заслонки выбранного источника
	_startPreheatingTimerTrigger:BOOL;//Триггер запуска таймера
	_startOpenQuartzTimerTrigger:BOOL;//Триггер запуска таймера ожидания при открытом кварцевом датчике
	_startQuartzSensoreHeatingTimerTrigger:BOOL;//Триггер запуска таймера прогрева кварцевого датчика 
	_commandLock:				BOOL;//Блокировка ввода новой комманды
	_InitDone:					BOOL;
	xInit:						BOOL;
END_VAR

{TODO:"Добавить начальную силу тока для старта"}
(*
[x]Проверка на нулевые значения указателей
[]Обработка датчика давления
[]Обработка всех ошибок исходя из статуса
*)

_preHeatTimer(IN:=_startPreheatingTimerTrigger,
				ET=>_preHeatLeftTime);
_qartzOpenDelayTimer(IN:=_startOpenQuartzTimerTrigger);
_qartzHeatingTimer(IN:=_startQuartzSensoreHeatingTimerTrigger);



THIS^.Update();				

CASE _stage OF
	DepositeProcessStage.WAIT_COMMAND:
		(*THIS^.Status:=GornDepositeProccessStatus.WAIT_COMMAND;
		IF  refStarProcess AND NOT _commandLock THEN
			refStarProcess:=FALSE;
			_commandLock:=TRUE;
			_stage:=DepositeProcessStage.INIT_DATA;
		ELSIF refStarProcess AND _commandLock THEN
			refStarProcess:=FALSE;
			_stage:=DepositeProcessStage.ERROR;
			THIS^.Status:=GornDepositeProccessStatus.COMMAND_LOCK;
			RETURN;
		END_IF*)
	DepositeProcessStage.INIT_DATA:
		(*//Уставка времени для таймеров
		InitTimers();
		//Выбор нужных устройств для напыления
		SelectDepositeSource();
		//Проверка на Nullptr
		IF _ptrGorn = 0 THEN
			_stage:=DepositeProcessStage.ERROR;
			Status:=GornDepositeProccessStatus.GORN_NULL_PTR;
			RETURN;
		END_IF
		IF _ptrQuartzRawRate = 0 THEN
			_stage:=DepositeProcessStage.ERROR;
			Status:=GornDepositeProccessStatus.QUARTZ_RAW_RATE_NULL_PTR;
			RETURN;			
		END_IF
		IF _ptrThinkness = 0 THEN
			_stage:=DepositeProcessStage.ERROR;
			Status:=GornDepositeProccessStatus.THINKNESS_NULL_PTR;
			RETURN;
		END_IF
		IF _ptrQuartzReset = 0 THEN
			_stage:=DepositeProcessStage.ERROR;
			Status:=GornDepositeProccessStatus.QUARTZ_RESET_NULL_PTR;
			RETURN;
		END_IF
		IF _ptrGornSetting = 0 THEN
			_stage:=DepositeProcessStage.ERROR;
			Status:=GornDepositeProccessStatus.GORN_SETTING_NULL_PTR;
			RETURN;
		END_IF
		IF _ptrShutter =0 THEN
			_stage:=DepositeProcessStage.ERROR;
			Status:=GornDepositeProccessStatus.SHUTTER_NULL_PTR;
			RETURN;
		END_IF
		IF _ptrShutterSetting = 0 THEN
			_stage:=DepositeProcessStage.ERROR;
			Status:=GornDepositeProccessStatus.SHUTTER_SETTING_NULL_PTR;
			RETURN;
		END_IF
		IF _ptrQuartzShutter = 0 THEN
			_stage:=DepositeProcessStage.ERROR;
			Status:=GornDepositeProccessStatus.QUARTZ_SHUTTER_NULL_PTR;
			RETURN;
		END_IF
		
		IF NOT _ptrGornSetting^.xAutoMode THEN
			_stage:=DepositeProcessStage.ERROR;
			Status:=GornDepositeProccessStatus.GORN_NOT_AUTOMODE;
			RETURN;
		END_IF
		IF NOT _ptrShutterSetting^.AutoMode THEN
			_stage:=DepositeProcessStage.ERROR;
			Status:=GornDepositeProccessStatus.SHUTTER_NOT_AUTOMODE;
			RETURN;
		END_IF
		IF NOT _ptrShutterSetting^.RemoteMode THEN
			_stage:=DepositeProcessStage.ERROR;
			Status:=GornDepositeProccessStatus.SHUTTER_LOCALMODE;
			RETURN;
		END_IF
		IF _ptrGorn^.xBlocked THEN
			_stage:=DepositeProcessStage.ERROR;
			Status:=GornDepositeProccessStatus.GORN_BLOCKED;
			RETURN;
		END_IF
		IF NOT _ptrGorn^.xPowerEnable THEN
			_stage:=DepositeProcessStage.ERROR;
			Status:=GornDepositeProccessStatus.GORN_NOT_POWER;
			RETURN;
		END_IF
		IF NOT _ptrGorn^.xModbusConnected THEN
			_stage:=DepositeProcessStage.ERROR;
			Status:=GornDepositeProccessStatus.GORN_OFFLINE;
			RETURN;
		END_IF
		
		
		refProcessData.iPreheatCurrent:=refProcessSetting.StartPreheatSP;
		refProcessSetting.PIDManualMode:=TRUE;
		_InitDone:=TRUE;
		Status:= GornDepositeProccessStatus.INIT_DONE;
		_stage:= DepositeProcessStage.START_HEATER;
		*)
	DepositeProcessStage.START_HEATER:
		(*_ptrGorn^.xAutoCommand:=TRUE;
		IF _ptrGorn^.xTurnOn THEN
			_startPreheatingTimerTrigger:=TRUE;
			Status:=GornDepositeProccessStatus.GORN_TURNON;
			_stage:=DepositeProcessStage.PREDEPOSITE_HEATING;
		END_IF
		IF _ptrGorn^.xError THEN
			_ptrGorn^.xAutoCommand:=FALSE;
			_startPreheatingTimerTrigger:=FALSE;
			Status:=GornDepositeProccessStatus.GORN_ERROR;
			_stage:=DepositeProcessStage.ERROR;
			RETURN;
		END_IF*)
		
 	DepositeProcessStage.PREDEPOSITE_HEATING:
// 		refProcessData.iPreheatCurrent:=CalcSP();
// 		_ptrGornSetting^.rSpCurrent:=refProcessData.iPreheatCurrent;
// 		IF _preHeatTimer.Q THEN
// 			Status:=GornDepositeProccessStatus.PREHEAT_DONE;
// 			_stage:=DepositeProcessStage.QARTZ_OPEN;
// 		END_IF
		
		//TODO: обработка аварийных ситуаций
 	DepositeProcessStage.QARTZ_OPEN:
// 		//TODO: Обработка ошибки по недостаточному давлению
// 		_ptrQuartzShutter^.xValue:=TRUE;
// 		_startOpenQuartzTimerTrigger:=TRUE;
// 		Status:=GornDepositeProccessStatus.QUARTZ_SHUTTER_OPENED;
// 		_stage:=DepositeProcessStage.QUARTZ_OPENED_DELAY;
// 		

	DepositeProcessStage.QUARTZ_OPENED_DELAY:
// 		IF _qartzOpenDelayTimer.Q THEN
// 			_stage:=DepositeProcessStage.SOURCE_SHUTTER_OPEN;
// 			Status:=GornDepositeProccessStatus.QUARTZ_DELAY_DONE;
// 		END_IF	
// 		
	DepositeProcessStage.SOURCE_SHUTTER_OPEN:
// 		_ptrShutter^.AutoCommand:=TRUE;
// 		IF _ptrShutter^.ShutterOpened THEN
// 			_startQuartzSensoreHeatingTimerTrigger:=TRUE;
// 			Status:=GornDepositeProccessStatus.SHUTTER_OPENED;
// 			_stage:=DepositeProcessStage.QARTZ_SENSORE_HEATING;
// 		END_IF
		
	DepositeProcessStage.QARTZ_SENSORE_HEATING:
// 		Status:=GornDepositeProccessStatus.QUARTZ_HEATING;
// 		IF _qartzHeatingTimer.Q THEN
// 			refProcessSetting.PIDManualMode:=FALSE;
// 			refProcessData.SPtoPID:=refProcessSetting.DepositeSpeedSP_1;
// 			_ptrQuartzReset^:=TRUE;
// 			Status:=GornDepositeProccessStatus.QUARTZ_HEATER;
// 			_stage:=DepositeProcessStage.LIMIT_SPEED_DEPOSITE_1;
// 		END_IF
	DepositeProcessStage.LIMIT_SPEED_DEPOSITE_1:
// 		_ptrGornSetting^.rSpCurrent:=refProcessData.iPreheatCurrent;
// 		refProcessData.rActualRawRate:=_ptrQuartzRawRate^;
// 		Status:=GornDepositeProccessStatus.FIRST_STAGE_DEPOSITE;
// 		IF _ptrThinkness^>=refProcessSetting.DepositeThinkness_1 THEN
// 			refProcessData.SPtoPID:=refProcessSetting.DepositeSpeedSP_2;
// 			_stage:=DepositeProcessStage.LIMIT_SPEED_DEPOSITE_2;
// 			Status:=GornDepositeProccessStatus.FIRST_STAGE_DEPOSITE_DONE;
// 		END_IF
		
	DepositeProcessStage.LIMIT_SPEED_DEPOSITE_2:
// 		_ptrGornSetting^.rSpCurrent:=refProcessData.iPreheatCurrent;
// 		refProcessData.rActualRawRate:=_ptrQuartzRawRate^;
// 		Status:=GornDepositeProccessStatus.SECOND_STAGE_DEPOSITE;
// 		IF _ptrThinkness^ >= refProcessSetting.DepositeThinkness_2 THEN
// 			_ptrShutter^.AutoCommand:=FALSE;
// 			_ptrQuartzShutter^.xValue:=FALSE;
// 			Status:=GornDepositeProccessStatus.SECOND_STAGE_DEPOSITE_DONE;
// 			_stage:=DepositeProcessStage.STOP_DEPOSITE;
// 		END_IF
		
	DepositeProcessStage.STOP_DEPOSITE:
// 		_ptrGorn^.xAutoCommand:=FALSE;
// 		refProcessSetting.PIDManualMode:=TRUE;
// 		refProcessData.iPreheatCurrent := refProcessSetting.StartPreheatSP;
// 		_ptrGornSetting^.rSpCurrent:=refProcessData.iPreheatCurrent;
// 		_commandLock:=FALSE;
// 		_InitDone:=FALSE;
// 		Status:=GornDepositeProccessStatus.STOP_DEPOSITE;
// 		_stage:=DepositeProcessStage.WAIT_COMMAND;
	DepositeProcessStage.ERROR:
// 		_ptrGorn^.xAutoCommand:=FALSE;
// 		refProcessSetting.PIDManualMode:=TRUE;
// 		_ptrQuartzShutter^.xValue:=FALSE;
// 		_ptrShutter^.AutoCommand:=FALSE;
// 		_InitDone:=FALSE;
// 		refProcessData.iPreheatCurrent := refProcessSetting.StartPreheatSP;
// 		_ptrGornSetting^.rSpCurrent:=refProcessData.iPreheatCurrent;
// 		IF refAcknowledgment THEN
// 			refAcknowledgment:=FALSE;
// 			_commandLock:=FALSE;
// 			_stage:=DepositeProcessStage.WAIT_COMMAND;
// 		END_IF
		
END_CASE

(*
Метод собирающий разрешение на запуск 
*)
METHOD AssemblePermition : WORD
VAR_INPUT
END_VAR
//Проверка на nullptr
IF THIS^.ptrGornList[THIS^.refProcessSetting.DepositeSourse] = 0 THEN
	AssemblePermition:=AssemblePermitionStatusList.GornPointerNullPtr;
	THIS^._permition:=FALSE;
	RETURN;
END_IF

IF THIS^.ptrShutterList[THIS^.refProcessSetting.DepositeSourse]=0 THEN
	AssemblePermition:=AssemblePermitionStatusList.ShutterPointerNullPtr;
	THIS^._permition:=FALSE;	
	RETURN; 
END_IF


//Разрешение выбранного горна
THIS^._selectedGornPermition:=	THIS^.ptrGornList[THIS^.refProcessSetting.DepositeSourse]^.xPowerEnable AND
								THIS^.ptrGornList[THIS^.refProcessSetting.DepositeSourse]^.xPowerOnFeedback AND 
								THIS^.ptrGornList[THIS^.refProcessSetting.DepositeSourse]^.xAutoMode AND
								THIS^.ptrGornList[THIS^.refProcessSetting.DepositeSourse]^.xModbusConnected AND
								NOT THIS^.ptrGornList[THIS^.refProcessSetting.DepositeSourse]^.xBlocked AND
								NOT THIS^.ptrGornList[THIS^.refProcessSetting.DepositeSourse]^.xError;
								
THIS^._selectedShutterPermition:=	NOT THIS^.ptrShutterList[THIS^.refProcessSetting.DepositeSourse]^.Interlock AND
									THIS^.ptrShutterList[THIS^.refProcessSetting.DepositeSourse]^.AutoMode;
END_METHOD

METHOD PRIVATE CalcSP : INT
VAR_INPUT
END_VAR
CalcSP:=(((refProcessSetting.FinallyPreheatSP-refProcessSetting.StartPreheatSP)/refProcessSetting.PreheatingTime)*getPreheatTimeLeftSecond)+refProcessSetting.StartPreheatSP;
END_METHOD

METHOD PRIVATE InitTimers
VAR_INPUT
END_VAR
_preHeatTimer.PT:=UINT_TO_TIME(refProcessSetting.PreheatingTime * 1000);
_qartzOpenDelayTimer.PT:=UINT_TO_TIME(THIS^.refProcessSetting.QuartzDelayTime *1000);
_qartzHeatingTimer.PT:=UINT_TO_TIME(THIS^.refProcessSetting.QuartzHeatingTime * 1000);
END_METHOD

METHOD SelectDepositeSource
VAR_INPUT
END_VAR
		_ptrGorn:=ptrGornList[refProcessSetting.DepositeSourse];
		_ptrShutter:=ptrShutterList[refProcessSetting.DepositeSourse];
		_ptrGornSetting:=ptrGornSettingList[refProcessSetting.DepositeSourse];
		_ptrShutterSetting:=ptrShutterSettingList[refProcessSetting.DepositeSourse];
		_ptrQuartzShutter:=ptrQuartzShutterList[refProcessSetting.DepositeSourse];
		_ptrQuartzReset:=ptrQuartzResetList[refProcessSetting.DepositeSourse];
		_ptrThinkness:=ptrThinknessList[refProcessSetting.DepositeSourse];
		_ptrQuartzRawRate:=ptrQuartzResetList[refProcessSetting.DepositeSourse];
END_METHOD

METHOD PRIVATE Update : WORD
VAR_INPUT
END_VAR
refProcessData.Stage:=_stage;
IF _InitDone THEN
	refProcessData.iMinRegValue:=_ptrGornSetting^.rMinSpCurrent;
	refProcessData.iMaxRegValue:=_ptrGornSetting^.rMaxSpCurrent;
	refProcessData.ActualThinkness:=_ptrThinkness^;
	refProcessData.iRegValueFB:=_ptrGorn^.rFbCurrent;
	RETURN;
END_IF
refProcessData.iMinRegValue:=0;
refProcessData.iMaxRegValue:=0;
END_METHOD

//Прошедшее время с момента запуска препрогрева
PROPERTY PRIVATE getPreheatTimeLeftSecond : UINT
GET
getPreheatTimeLeftSecond:=DWORD_TO_UINT(TIME_TO_DWORD(THIS^._preheatLeftTime)/1000);
END_GET
END_PROPERTY

PROPERTY setGorn1 : DINT
SET
THIS^.ptrGornList[0]:= setGorn1;
END_SET
END_PROPERTY

PROPERTY setGorn2 : DINT
SET
THIS^.ptrGornList[1]:=setGorn2;
END_SET
END_PROPERTY

PROPERTY setGorn3 : DINT
SET
THIS^.ptrGornList[2]:=setGorn3;
END_SET
END_PROPERTY

PROPERTY setGornSetting1 : DINT
SET
THIS^.ptrGornSettingList[0]:=setGornSetting1;
END_SET
END_PROPERTY

PROPERTY setGornSetting2 : DINT
SET
THIS^.ptrGornSettingList[1]:=setGornSetting2;
END_SET
END_PROPERTY

PROPERTY setGornSetting3 : DINT
SET
THIS^.ptrGornSettingList[2]:=setGornSetting3;
END_SET
END_PROPERTY

PROPERTY setQartzReset1 : DINT
SET
THIS^.ptrQuartzResetList[0]:=setQartzReset1;
END_SET
END_PROPERTY

PROPERTY setQartzReset2 : DINT
SET
THIS^.ptrQuartzResetList[1]:=setQartzReset2;
END_SET
END_PROPERTY

PROPERTY setQartzReset3 : DINT
SET
THIS^.ptrQuartzResetList[2]:=setQartzReset3;
END_SET
END_PROPERTY

PROPERTY setQuartzShutter1 : DINT
SET
THIS^.ptrQuartzShutterList[0]:=setQuartzShutter1;
END_SET
END_PROPERTY

PROPERTY setQuartzShutter2 : DINT
SET
THIS^.ptrQuartzShutterList[1]:=setQuartzShutter2;
END_SET
END_PROPERTY

PROPERTY setQuartzShutter3 : DINT
SET
THIS^.ptrQuartzShutterList[2]:=setQuartzShutter3;
END_SET
END_PROPERTY

PROPERTY setRawRate1 : DINT
SET
ptrMaterialRawRateList[0]:=setRawRate1;
END_SET
END_PROPERTY

PROPERTY setRawRate2 : DINT
SET
ptrMaterialRawRateList[1]:=setRawRate2;
END_SET
END_PROPERTY

PROPERTY setRawRate3 : DINT
SET
ptrMaterialRawRateList[2]:=setRawRate3;
END_SET
END_PROPERTY

PROPERTY setShutter1 : DINT
SET
THIS^.ptrShutterList[0]:=setShutter1;
END_SET
END_PROPERTY

PROPERTY setShutter2 : DINT
SET
THIS^.ptrShutterList[1]:=setShutter2;
END_SET
END_PROPERTY

PROPERTY setShutter3 : DINT
SET
THIS^.ptrShutterList[2]:=setShutter3;
END_SET
END_PROPERTY

PROPERTY setShutterSetting1 : DINT
SET
THIS^.ptrShutterSettingList[0]:=setShutterSetting1;
END_SET
END_PROPERTY

PROPERTY setShutterSetting2 : DINT
SET
THIS^.ptrShutterSettingList[1]:=setShutterSetting2;
END_SET
END_PROPERTY

PROPERTY setShutterSetting3 : DINT
SET
THIS^.ptrShutterSettingList[2]:=setShutterSetting3;
END_SET
END_PROPERTY

PROPERTY setThinkness1 : DINT
SET
THIS^.ptrThinknessList[0]:=setThinkness1;
END_SET
END_PROPERTY

PROPERTY setThinkness2 : DINT
SET
THIS^.ptrThinknessList[1]:=setThinkness2;
END_SET
END_PROPERTY

PROPERTY setThinkness3 : DINT
SET
THIS^.ptrThinknessList[2]:=setThinkness3;
END_SET
END_PROPERTY

END_FUNCTION_BLOCK

// Function Blocks/DepositeProccess/fbGornDepositeProccess
FUNCTION_BLOCK fbGornDepositeProccess
VAR_INPUT
	refStarProcess:				REFERENCE TO BOOL; //Команда на старт процесса
	refAcknowledgment:			REFERENCE TO BOOL; //команда на сброс ошибки.
	refStopCommand:				REFERENCE TO BOOL; //Команда на остановку процесса
	refProcessSetting: 			REFERENCE TO udtGornDepositeProccessSetting;
	refProcessData:	   			REFERENCE TO udtGornDepositeProccessData;
END_VAR
VAR_OUTPUT
	Status :					WORD;
END_VAR
VAR
	ptrGornList: 				ARRAY[0..2] OF POINTER TO udtGorn;
	ptrGornSettingList:			ARRAY[0..2] OF POINTER TO udtGornSetting;
	ptrShutterList:				ARRAY[0..2] OF POINTER TO udtShutter;
	ptrShutterSettingList:		ARRAY[0..2] OF POINTER TO udtShutterSetting;
	ptrQuartzShutterList:		ARRAY[0..2] OF POINTER TO udtDiscreteSignal;
	ptrQuartzResetList:			ARRAY[0..2] OF POINTER TO BOOL;
	ptrThinknessList:			ARRAY[0..2] OF POINTER TO REAL;
	ptrMaterialRawRateList:		ARRAY[0..2] OF POINTER TO REAL;
	_ptrGorn:					POINTER TO udtGorn;
	_ptrGornSetting:			POINTER TO udtGornSetting;
	_ptrShutter:				POINTER TO udtShutter;
	_ptrShutterSetting:			POINTER TO udtShutterSetting;
	_ptrQuartzShutter:			POINTER TO udtDiscreteSignal;
	_ptrQuartzReset:			POINTER TO BOOL;
	_ptrThinkness:				POINTER TO REAL;
	_ptrQuartzRawRate:			POINTER TO REAL;
	_preHeatTimer:				TON;//Время препрогрева
	_preheatLeftTime:			TIME;//(мс)Прошедшее время с момента препрогрева
	
	_qartzOpenDelayTimer:		TON;//Время открытия кварцевого датчика до напыления
	_qartzHeatingTimer:			TON;//Время прогрева кварцевого датчика
	_assemblePermitionStatus:	WORD;
	_stage:						INT; //Стадии работы
	
	_permition:					BOOL;//Разрешение на старт процесса
	_selectedGornPermition: 	BOOL;//Разрешение на старт выбранного источника тока
	_selectedShutterPermition:	BOOL;//Разрешение от заслонки выбранного источника
	_startPreheatingTimerTrigger:BOOL;//Триггер запуска таймера
	_startOpenQuartzTimerTrigger:BOOL;//Триггер запуска таймера ожидания при открытом кварцевом датчике
	_startQuartzSensoreHeatingTimerTrigger:BOOL;//Триггер запуска таймера прогрева кварцевого датчика 
	_commandLock:				BOOL;//Блокировка ввода новой комманды
	_InitDone:					BOOL;
	xInit:						BOOL;
END_VAR

{TODO:"Добавить начальную силу тока для старта"}
(*
[x]Проверка на нулевые значения указателей
[]Обработка датчика давления
[]Обработка всех ошибок исходя из статуса
*)

_preHeatTimer(IN:=_startPreheatingTimerTrigger,
				ET=>_preHeatLeftTime);
_qartzOpenDelayTimer(IN:=_startOpenQuartzTimerTrigger);
_qartzHeatingTimer(IN:=_startQuartzSensoreHeatingTimerTrigger);



THIS^.Update();	
IF refStopCommand THEN
	refStopCommand:=FALSE;
	_stage:=DepositeProcessStage.STOP_DEPOSITE;
END_IF			

CASE _stage OF
	DepositeProcessStage.WAIT_COMMAND:
		THIS^.Status:=GornDepositeProccessStatus.WAIT_COMMAND;
		IF  refStarProcess AND NOT _commandLock THEN
			refStarProcess:=FALSE;
			_commandLock:=TRUE;
			_stage:=DepositeProcessStage.INIT_DATA;
		ELSIF refStarProcess AND _commandLock THEN
			refStarProcess:=FALSE;
			_stage:=DepositeProcessStage.ERROR;
			THIS^.Status:=GornDepositeProccessStatus.COMMAND_LOCK;
			RETURN;
		END_IF
	DepositeProcessStage.INIT_DATA:
		//Уставка времени для таймеров
		InitTimers();
		//Выбор нужных устройств для напыления
		SelectDepositeSource();
		//Проверка на Nullptr
		IF _ptrGorn = 0 THEN
			_stage:=DepositeProcessStage.ERROR;
			Status:=GornDepositeProccessStatus.GORN_NULL_PTR;
			RETURN;
		END_IF
		IF _ptrQuartzRawRate = 0 THEN
			_stage:=DepositeProcessStage.ERROR;
			Status:=GornDepositeProccessStatus.QUARTZ_RAW_RATE_NULL_PTR;
			RETURN;			
		END_IF
		IF _ptrThinkness = 0 THEN
			_stage:=DepositeProcessStage.ERROR;
			Status:=GornDepositeProccessStatus.THINKNESS_NULL_PTR;
			RETURN;
		END_IF
		IF _ptrQuartzReset = 0 THEN
			_stage:=DepositeProcessStage.ERROR;
			Status:=GornDepositeProccessStatus.QUARTZ_RESET_NULL_PTR;
			RETURN;
		END_IF
		IF _ptrGornSetting = 0 THEN
			_stage:=DepositeProcessStage.ERROR;
			Status:=GornDepositeProccessStatus.GORN_SETTING_NULL_PTR;
			RETURN;
		END_IF
		IF _ptrShutter =0 THEN
			_stage:=DepositeProcessStage.ERROR;
			Status:=GornDepositeProccessStatus.SHUTTER_NULL_PTR;
			RETURN;
		END_IF
		IF _ptrShutterSetting = 0 THEN
			_stage:=DepositeProcessStage.ERROR;
			Status:=GornDepositeProccessStatus.SHUTTER_SETTING_NULL_PTR;
			RETURN;
		END_IF
		IF _ptrQuartzShutter = 0 THEN
			_stage:=DepositeProcessStage.ERROR;
			Status:=GornDepositeProccessStatus.QUARTZ_SHUTTER_NULL_PTR;
			RETURN;
		END_IF
		
		IF NOT _ptrGornSetting^.xAutoMode THEN
			_stage:=DepositeProcessStage.ERROR;
			Status:=GornDepositeProccessStatus.GORN_NOT_AUTOMODE;
			RETURN;
		END_IF
		IF NOT _ptrShutterSetting^.AutoMode THEN
			_stage:=DepositeProcessStage.ERROR;
			Status:=GornDepositeProccessStatus.SHUTTER_NOT_AUTOMODE;
			RETURN;
		END_IF
		IF NOT _ptrShutterSetting^.RemoteMode THEN
			_stage:=DepositeProcessStage.ERROR;
			Status:=GornDepositeProccessStatus.SHUTTER_LOCALMODE;
			RETURN;
		END_IF
		IF _ptrGorn^.xBlocked THEN
			_stage:=DepositeProcessStage.ERROR;
			Status:=GornDepositeProccessStatus.GORN_BLOCKED;
			RETURN;
		END_IF
		IF NOT _ptrGorn^.xPowerEnable THEN
			_stage:=DepositeProcessStage.ERROR;
			Status:=GornDepositeProccessStatus.GORN_NOT_POWER;
			RETURN;
		END_IF
		IF NOT _ptrGorn^.xModbusConnected THEN
			_stage:=DepositeProcessStage.ERROR;
			Status:=GornDepositeProccessStatus.GORN_OFFLINE;
			RETURN;
		END_IF
		
		
		refProcessData.iPreheatCurrent:=refProcessSetting.StartPreheatSP;
		_ptrGornSetting^.rAutoModeCurrent:=refProcessSetting.StartPreheatSP;
		refProcessSetting.PIDManualMode:=TRUE;
		_InitDone:=TRUE;
		Status:= GornDepositeProccessStatus.INIT_DONE;
		_stage:= DepositeProcessStage.START_HEATER;
		_ptrGorn^.xAutoPowerCommand:=TRUE;
	DepositeProcessStage.START_HEATER:
		_ptrGorn^.xAutoCommand:=TRUE;
		IF _ptrGorn^.xTurnOn THEN
			_startPreheatingTimerTrigger:=TRUE;
			Status:=GornDepositeProccessStatus.GORN_TURNON;
			_stage:=DepositeProcessStage.PREDEPOSITE_HEATING;
		END_IF
		IF _ptrGorn^.xError THEN
			_ptrGorn^.xAutoCommand:=FALSE;
			_startPreheatingTimerTrigger:=FALSE;
			Status:=GornDepositeProccessStatus.GORN_ERROR;
			_stage:=DepositeProcessStage.ERROR;
			RETURN;
		END_IF
	DepositeProcessStage.PREDEPOSITE_HEATING:
		refProcessData.iPreheatCurrent:=CalcSP();
		_ptrGornSetting^.rAutoModeCurrent:=refProcessData.iPreheatCurrent;
		IF _preHeatTimer.Q THEN
			Status:=GornDepositeProccessStatus.PREHEAT_DONE;
			_stage:=DepositeProcessStage.QARTZ_OPEN;
		END_IF
		//TODO: обработка аварийных ситуаций
	DepositeProcessStage.QARTZ_OPEN:
		//TODO: Обработка ошибки по недостаточному давлению
		_ptrQuartzShutter^.xValue:=TRUE;
		_startOpenQuartzTimerTrigger:=TRUE;
		Status:=GornDepositeProccessStatus.QUARTZ_SHUTTER_OPENED;
		_stage:=DepositeProcessStage.QUARTZ_OPENED_DELAY;
		
	DepositeProcessStage.QUARTZ_OPENED_DELAY:
		IF _qartzOpenDelayTimer.Q THEN
			_stage:=DepositeProcessStage.SOURCE_SHUTTER_OPEN;
			Status:=GornDepositeProccessStatus.QUARTZ_DELAY_DONE;
		END_IF	
		
	DepositeProcessStage.SOURCE_SHUTTER_OPEN:
		_ptrShutter^.AutoCommand:=TRUE;
		IF _ptrShutter^.ShutterOpened THEN
			_startQuartzSensoreHeatingTimerTrigger:=TRUE;
			Status:=GornDepositeProccessStatus.SHUTTER_OPENED;
			_stage:=DepositeProcessStage.QARTZ_SENSORE_HEATING;
		END_IF
		
	DepositeProcessStage.QARTZ_SENSORE_HEATING:
		Status:=GornDepositeProccessStatus.QUARTZ_HEATING;
		IF _qartzHeatingTimer.Q THEN
			refProcessSetting.PIDManualMode:=FALSE;
			refProcessData.SPtoPID:=refProcessSetting.DepositeSpeedSP_1;
			_ptrQuartzReset^:=TRUE;
			Status:=GornDepositeProccessStatus.QUARTZ_HEATER;
			_stage:=DepositeProcessStage.LIMIT_SPEED_DEPOSITE_1;
		END_IF
	DepositeProcessStage.LIMIT_SPEED_DEPOSITE_1:
		_ptrGornSetting^.rSpCurrent:=refProcessData.iPreheatCurrent;
		refProcessData.rActualRawRate:=_ptrQuartzRawRate^;
		Status:=GornDepositeProccessStatus.FIRST_STAGE_DEPOSITE;
		IF _ptrThinkness^>=refProcessSetting.DepositeThinkness_1 THEN
			refProcessData.SPtoPID:=refProcessSetting.DepositeSpeedSP_2;
			_stage:=DepositeProcessStage.LIMIT_SPEED_DEPOSITE_2;
			Status:=GornDepositeProccessStatus.FIRST_STAGE_DEPOSITE_DONE;
		END_IF
		
	DepositeProcessStage.LIMIT_SPEED_DEPOSITE_2:
		_ptrGornSetting^.rSpCurrent:=refProcessData.iPreheatCurrent;
		refProcessData.rActualRawRate:=_ptrQuartzRawRate^;
		Status:=GornDepositeProccessStatus.SECOND_STAGE_DEPOSITE;
		IF _ptrThinkness^ >= refProcessSetting.DepositeThinkness_2 THEN
			_ptrShutter^.AutoCommand:=FALSE;
			_ptrQuartzShutter^.xValue:=FALSE;
			Status:=GornDepositeProccessStatus.SECOND_STAGE_DEPOSITE_DONE;
			_stage:=DepositeProcessStage.STOP_DEPOSITE;
		END_IF
		
	DepositeProcessStage.STOP_DEPOSITE:
		_ptrGorn^.xAutoCommand:=FALSE;
		refProcessSetting.PIDManualMode:=TRUE;
		refProcessData.iPreheatCurrent := refProcessSetting.StartPreheatSP;
		_ptrGornSetting^.rSpCurrent:=refProcessData.iPreheatCurrent;
		_commandLock:=FALSE;
		_InitDone:=FALSE;
		_ptrQuartzShutter^.xValue:=FALSE;
		_ptrShutter^.AutoCommand:=FALSE;
		Status:=GornDepositeProccessStatus.STOP_DEPOSITE;
		_stage:=DepositeProcessStage.WAIT_COMMAND;
		_startPreheatingTimerTrigger:=FALSE;
		_startOpenQuartzTimerTrigger:=FALSE;
		_startQuartzSensoreHeatingTimerTrigger:=FALSE;
	DepositeProcessStage.ERROR:
		_ptrGorn^.xAutoCommand:=FALSE;
		refProcessSetting.PIDManualMode:=TRUE;
		_ptrQuartzShutter^.xValue:=FALSE;
		_ptrShutter^.AutoCommand:=FALSE;
		_InitDone:=FALSE;
		refProcessData.iPreheatCurrent := refProcessSetting.StartPreheatSP;
		_ptrGornSetting^.rSpCurrent:=refProcessData.iPreheatCurrent;
		_startPreheatingTimerTrigger:=FALSE;
		_startOpenQuartzTimerTrigger:=FALSE;
		_startQuartzSensoreHeatingTimerTrigger:=FALSE;
		IF refAcknowledgment THEN
			refAcknowledgment:=FALSE;
			_commandLock:=FALSE;
			_stage:=DepositeProcessStage.WAIT_COMMAND;
		END_IF
		
END_CASE
refProcessData.Stage:=_stage;
refProcessData.ActualThinkness:=_ptrThinkness^;

(*
Метод собирающий разрешение на запуск 
*)
METHOD AssemblePermition : WORD
VAR_INPUT
END_VAR
//Проверка на nullptr
IF THIS^.ptrGornList[THIS^.refProcessSetting.DepositeSourse] = 0 THEN
	AssemblePermition:=AssemblePermitionStatusList.GornPointerNullPtr;
	THIS^._permition:=FALSE;
	RETURN;
END_IF

IF THIS^.ptrShutterList[THIS^.refProcessSetting.DepositeSourse]=0 THEN
	AssemblePermition:=AssemblePermitionStatusList.ShutterPointerNullPtr;
	THIS^._permition:=FALSE;	
	RETURN; 
END_IF


//Разрешение выбранного горна
THIS^._selectedGornPermition:=	THIS^.ptrGornList[THIS^.refProcessSetting.DepositeSourse]^.xPowerEnable AND
								THIS^.ptrGornList[THIS^.refProcessSetting.DepositeSourse]^.xPowerOnFeedback AND 
								THIS^.ptrGornList[THIS^.refProcessSetting.DepositeSourse]^.xAutoMode AND
								THIS^.ptrGornList[THIS^.refProcessSetting.DepositeSourse]^.xModbusConnected AND
								NOT THIS^.ptrGornList[THIS^.refProcessSetting.DepositeSourse]^.xBlocked AND
								NOT THIS^.ptrGornList[THIS^.refProcessSetting.DepositeSourse]^.xError;
								
THIS^._selectedShutterPermition:=	NOT THIS^.ptrShutterList[THIS^.refProcessSetting.DepositeSourse]^.Interlock AND
									THIS^.ptrShutterList[THIS^.refProcessSetting.DepositeSourse]^.AutoMode;
END_METHOD

METHOD PRIVATE CalcSP : INT
VAR_INPUT
END_VAR
CalcSP:=(((refProcessSetting.FinallyPreheatSP-refProcessSetting.StartPreheatSP)/refProcessSetting.PreheatingTime)*getPreheatTimeLeftSecond)+refProcessSetting.StartPreheatSP;
END_METHOD

METHOD PRIVATE InitTimers
VAR_INPUT
END_VAR
_preHeatTimer.PT:=UINT_TO_TIME(refProcessSetting.PreheatingTime * 1000);
_qartzOpenDelayTimer.PT:=UINT_TO_TIME(THIS^.refProcessSetting.QuartzDelayTime *1000);
_qartzHeatingTimer.PT:=UINT_TO_TIME(THIS^.refProcessSetting.QuartzHeatingTime * 1000);
END_METHOD

METHOD SelectDepositeSource
VAR_INPUT
END_VAR
		_ptrGorn:=ptrGornList[refProcessSetting.DepositeSourse];
		_ptrShutter:=ptrShutterList[refProcessSetting.DepositeSourse];
		_ptrGornSetting:=ptrGornSettingList[refProcessSetting.DepositeSourse];
		_ptrShutterSetting:=ptrShutterSettingList[refProcessSetting.DepositeSourse];
		_ptrQuartzShutter:=ptrQuartzShutterList[refProcessSetting.DepositeSourse];
		_ptrQuartzReset:=ptrQuartzResetList[refProcessSetting.DepositeSourse];
		_ptrThinkness:=ptrThinknessList[refProcessSetting.DepositeSourse];
		_ptrQuartzRawRate:=ptrQuartzResetList[refProcessSetting.DepositeSourse];
END_METHOD

METHOD PRIVATE Update : WORD
VAR_INPUT
END_VAR
refProcessData.Stage:=_stage;
IF _InitDone THEN
	refProcessData.iMinRegValue:=_ptrGornSetting^.rMinSpCurrent;
	refProcessData.iMaxRegValue:=_ptrGornSetting^.rMaxSpCurrent;
	refProcessData.ActualThinkness:=_ptrThinkness^;
	refProcessData.iRegValueFB:=_ptrGorn^.rFbCurrent;
	RETURN;
END_IF
refProcessData.iMinRegValue:=10;
refProcessData.iMaxRegValue:=150;
END_METHOD

//Прошедшее время с момента запуска препрогрева
PROPERTY PRIVATE getPreheatTimeLeftSecond : UINT
GET
getPreheatTimeLeftSecond:=DWORD_TO_UINT(TIME_TO_DWORD(THIS^._preheatLeftTime)/1000);
END_GET
END_PROPERTY

PROPERTY setGorn1 : DINT
SET
THIS^.ptrGornList[0]:= setGorn1;
END_SET
END_PROPERTY

PROPERTY setGorn2 : DINT
SET
THIS^.ptrGornList[1]:=setGorn2;
END_SET
END_PROPERTY

PROPERTY setGorn3 : DINT
SET
THIS^.ptrGornList[2]:=setGorn3;
END_SET
END_PROPERTY

PROPERTY setGornSetting1 : DINT
SET
THIS^.ptrGornSettingList[0]:=setGornSetting1;
END_SET
END_PROPERTY

PROPERTY setGornSetting2 : DINT
SET
THIS^.ptrGornSettingList[1]:=setGornSetting2;
END_SET
END_PROPERTY

PROPERTY setGornSetting3 : DINT
SET
THIS^.ptrGornSettingList[2]:=setGornSetting3;
END_SET
END_PROPERTY

PROPERTY setQartzReset1 : DINT
SET
THIS^.ptrQuartzResetList[0]:=setQartzReset1;
END_SET
END_PROPERTY

PROPERTY setQartzReset2 : DINT
SET
THIS^.ptrQuartzResetList[1]:=setQartzReset2;
END_SET
END_PROPERTY

PROPERTY setQartzReset3 : DINT
SET
THIS^.ptrQuartzResetList[2]:=setQartzReset3;
END_SET
END_PROPERTY

PROPERTY setQuartzShutter1 : DINT
SET
THIS^.ptrQuartzShutterList[0]:=setQuartzShutter1;
END_SET
END_PROPERTY

PROPERTY setQuartzShutter2 : DINT
SET
THIS^.ptrQuartzShutterList[1]:=setQuartzShutter2;
END_SET
END_PROPERTY

PROPERTY setQuartzShutter3 : DINT
SET
THIS^.ptrQuartzShutterList[2]:=setQuartzShutter3;
END_SET
END_PROPERTY

PROPERTY setRawRate1 : DINT
SET
ptrMaterialRawRateList[0]:=setRawRate1;
END_SET
END_PROPERTY

PROPERTY setRawRate2 : DINT
SET
ptrMaterialRawRateList[1]:=setRawRate2;
END_SET
END_PROPERTY

PROPERTY setRawRate3 : DINT
SET
ptrMaterialRawRateList[2]:=setRawRate3;
END_SET
END_PROPERTY

PROPERTY setShutter1 : DINT
SET
THIS^.ptrShutterList[0]:=setShutter1;
END_SET
END_PROPERTY

PROPERTY setShutter2 : DINT
SET
THIS^.ptrShutterList[1]:=setShutter2;
END_SET
END_PROPERTY

PROPERTY setShutter3 : DINT
SET
THIS^.ptrShutterList[2]:=setShutter3;
END_SET
END_PROPERTY

PROPERTY setShutterSetting1 : DINT
SET
THIS^.ptrShutterSettingList[0]:=setShutterSetting1;
END_SET
END_PROPERTY

PROPERTY setShutterSetting2 : DINT
SET
THIS^.ptrShutterSettingList[1]:=setShutterSetting2;
END_SET
END_PROPERTY

PROPERTY setShutterSetting3 : DINT
SET
THIS^.ptrShutterSettingList[2]:=setShutterSetting3;
END_SET
END_PROPERTY

PROPERTY setThinkness1 : DINT
SET
THIS^.ptrThinknessList[0]:=setThinkness1;
END_SET
END_PROPERTY

PROPERTY setThinkness2 : DINT
SET
THIS^.ptrThinknessList[1]:=setThinkness2;
END_SET
END_PROPERTY

PROPERTY setThinkness3 : DINT
SET
THIS^.ptrThinknessList[2]:=setThinkness3;
END_SET
END_PROPERTY

END_FUNCTION_BLOCK

// Function Blocks/DepositeProccess/GornDepositeUnit
FUNCTION_BLOCK GornDepositeUnit EXTENDS absDepositeUnit
VAR_INPUT
END_VAR
VAR_OUTPUT
END_VAR
VAR
	Device: POINTER TO udtGorn;
	DeviceSetting:	POINTER TO udtGornSetting;
END_VAR

METHOD   _addDepositeDevice : dpResult
VAR_INPUT
	ptrDevice	: 			POINTER TO BYTE;
	ptrDeviceSetting	: 	POINTER TO BYTE;
END_VAR
THIS^.Device:=ptrDevice;
THIS^.DeviceSetting:=ptrDeviceSetting;
END_METHOD

METHOD PROTECTED  _deviceAutoMode : BOOL
VAR_INPUT
END_VAR
_deviceAutoMode:=THIS^.Device^.xAutoMode;
END_METHOD

METHOD PROTECTED  _deviceManipulatingVariableGet : REAL
VAR_INPUT
END_VAR
_deviceManipulatingVariableGet:=TO_REAL(THIS^.DeviceSetting^.rAutoModeCurrent);
END_METHOD

METHOD PROTECTED  _deviceManipulatingVariableSet : dpResult
VAR_INPUT
	Variable: REAL;
END_VAR
THIS^.DeviceSetting^.rAutoModeCurrent:=TO_INT(Variable);
END_METHOD

METHOD PROTECTED  _maxManipulatingVariable : REAL
VAR_INPUT
END_VAR
_maxManipulatingVariable:=TO_REAL(THIS^.DeviceSetting^.rMaxSpCurrent);
END_METHOD

METHOD PROTECTED  _minManipulatingVariable : REAL
VAR_INPUT
END_VAR
_minManipulatingVariable:=TO_REAL(THIS^.DeviceSetting^.rMinSpCurrent);
END_METHOD

METHOD PROTECTED  _startDepositeDevice : dpResult
VAR_INPUT
	wStatus	: REFERENCE TO dpuStatus;
END_VAR
_startDepositeDevice:=DepositeResult.BUSY;
THIS^.Device^.xAutoCommand:=TRUE;
THIS^.Device^.xAutoPowerCommand:=TRUE;
IF THIS^.Device^.xTurnOn THEN
	wStatus:=DepositeProcessStatus.DEPOSITE_DEVICE_START;
	_startDepositeDevice:=DepositeResult.COMPLETE;
END_IF
END_METHOD

METHOD PROTECTED  _stopDepositeDevice : dpResult
VAR_INPUT
	wStatus	: REFERENCE TO dpuStatus;
END_VAR
_stopDepositeDevice:=DepositeResult.BUSY;
THIS^.Device^.xAutoCommand:=FALSE;
THIS^.Device^.xAutoPowerCommand:=FALSE;
IF NOT THIS^.Device^.xTurnOn THEN
	wStatus:=DepositeProcessStatus.DEPOSITE_DEVICE_STOP;
	_stopDepositeDevice:=DepositeResult.COMPLETE;
END_IF
END_METHOD

END_FUNCTION_BLOCK

// Function Blocks/DepositeProccess/HeaterDepositeUnit
FUNCTION_BLOCK HeaterDepositeUnit EXTENDS absDepositeUnit
VAR_INPUT
END_VAR
VAR_OUTPUT
END_VAR
VAR
	Device: POINTER TO udtHeater;
	DeviceSetting: POINTER TO udtHeaterSetting;
END_VAR

METHOD   _addDepositeDevice : dpResult
VAR_INPUT
	ptrDevice	: 			POINTER TO BYTE;
	ptrDeviceSetting	: 	POINTER TO BYTE;
END_VAR
_addDepositeDevice:=DepositeResult.BUSY;
THIS^.Device:=ptrDevice;
THIS^.DeviceSetting:=ptrDeviceSetting;
_addDepositeDevice:=DepositeResult.COMPLETE;
END_METHOD

METHOD PROTECTED  _deviceAutoMode : BOOL
VAR_INPUT
END_VAR
_deviceAutoMode:=THIS^.DeviceSetting^.xAutoMode;
END_METHOD

METHOD PROTECTED  _deviceManipulatingVariableGet : REAL
VAR_INPUT
END_VAR
_deviceManipulatingVariableGet:=THIS^.DeviceSetting^.rSetpointTemperature;
END_METHOD

METHOD PROTECTED  _deviceManipulatingVariableSet : dpResult
VAR_INPUT
	Variable: REAL;
END_VAR
THIS^.DeviceSetting^.rSetpointTemperature:=Variable;
END_METHOD

METHOD PROTECTED  _maxManipulatingVariable : REAL
VAR_INPUT
END_VAR
_maxManipulatingVariable:=THIS^.DeviceSetting^.rMaxPower;
END_METHOD

METHOD PROTECTED  _minManipulatingVariable : REAL
VAR_INPUT
END_VAR
_minManipulatingVariable:=THIS^.DeviceSetting^.rMinPower;
END_METHOD

METHOD PROTECTED  _startDepositeDevice : dpResult
VAR_INPUT
	wStatus	: REFERENCE TO dpuStatus;
END_VAR
_startDepositeDevice:=DepositeResult.BUSY;
THIS^.Device^.xAutoCommand:=TRUE;
IF THIS^.Device^.xPowerOn THEN
	_startDepositeDevice:=DepositeResult.COMPLETE;
	wStatus:=DepositeProcessStatus.DEPOSITE_DEVICE_START;
END_IF
END_METHOD

METHOD PROTECTED  _stopDepositeDevice : dpResult
VAR_INPUT
	wStatus	: REFERENCE TO dpuStatus;
END_VAR
_startDepositeDevice:=DepositeResult.BUSY;
THIS^.Device^.xAutoCommand:=FALSE;
IF NOT THIS^.Device^.xPowerOn THEN
	_startDepositeDevice:=DepositeResult.COMPLETE;
	wStatus:=DepositeProcessStatus.DEPOSITE_DEVICE_STOP;
END_IF
END_METHOD

END_FUNCTION_BLOCK

// Function Blocks/Driver/fbBSDDriver
FUNCTION_BLOCK fbBSDDriver
VAR_INPUT
	Driver:		REFERENCE TO udtBSDDriver;
	Setting:	REFERENCE TO udtBSDDriverSetting;
	Interlock:	BOOL;
	AlarmStop:	BOOL;
END_VAR
VAR_OUTPUT
	SpeedSignal:		UINT;
	StartSignal:		BOOL;
	CCWSignal:			BOOL;
	Run: 		BOOL;
	Blocked: 	BOOL;
END_VAR
VAR
END_VAR

IF AlarmStop THEN
	StartSignal:=FALSE;
	Run:=FALSE;
	Driver.xStartSignal := FALSE;
	RETURN;
END_IF



Driver.ServiceMode:=Setting.xServiceMode;
Driver.AutoMode:=Setting.xAutoMode;
Driver.xCCWSignal := Setting.xCCWMode;


IF Interlock AND NOT Setting.xServiceMode THEN
	Driver.Blocked := TRUE;
ELSE
	Driver.Blocked:=FALSE;
END_IF

IF Driver.AutoMode THEN
	Driver.xManualCommand:=Driver.xAutoCommand;
	Driver.rSpeedSP:= Setting.rAutoSpeedSP;
	Driver.xStartSignal:=Driver.xAutoCommand;
END_IF

IF NOT Driver.AutoMode THEN
	Driver.xAutoCommand := Driver.xManualCommand;
	Driver.rSpeedSP:=	Setting.rManualSpeedSP;
	Driver.xStartSignal:=Driver.xManualCommand;
END_IF

IF Driver.Blocked THEN
	Driver.xStartSignal:= FALSE;
END_IF


Driver.Run:=(Driver.xStartSignal AND Driver.rSpeedSP >0.0);


Driver.rSpeedSP:=LIMIT(0.0, Driver.rSpeedSP, Setting.rMaxSpeed);
StartSignal:=Driver.xStartSignal;
CCWSignal:=Driver.xCCWSignal;
Run:=Driver.Run;
Blocked:=Driver.Blocked;
SpeedSignal:=REAL_TO_UINT(Driver.rSpeedSP);

END_FUNCTION_BLOCK

// Function Blocks/GasRegulator/fbGasRegulator
FUNCTION_BLOCK fbGasRegulator
VAR_INPUT
	Setting: REFERENCE TO udtPIDSetting;
	CameraPressure:	REAL;
END_VAR
VAR_OUTPUT
	RRG1AutoSP: 	REAL;
	RRG2AutoSP:		REAL;
	RRG3AutoSP:		REAL;
	LimitsActive:	BOOL;
	OverFlow:		BOOL;
END_VAR
VAR
	PIDResult:REAL;
	Regulator: Util.PID;
END_VAR

Regulator(ACTUAL:=CameraPressure,
			SET_POINT:=Setting.rAutoSP,
			KP:=Setting.iP,
			TN:=Setting.tI,
			TV:=0.0,
			Y_MANUAL:=Setting.rMaunalSP,
			Y_OFFSET:=0.0,
			Y_MIN:=Setting.rMinSP,
			Y_MAX:=Setting.rMaxSP,
			MANUAL:=Setting.xAutoMode,
			RESET:=FALSE,
			Y=>PIDResult,
			LIMITS_ACTIVE=>LimitsActive,
			OVERFLOW=>OverFlow);
 
			
RRG1AutoSP:=CalcRRGSPwithCoeff(	V:=PIDResult,
								K:=Setting.rK1RRG);
								

RRG2AutoSP:=CalcRRGSPwithCoeff(	V:=PIDResult,
								K:=Setting.rK2RRG);
								

RRG3AutoSP:=CalcRRGSPwithCoeff(	V:=PIDResult,
								K:=Setting.rK3RRG);

METHOD CalcRRGSPwithCoeff : REAL
VAR_INPUT
	V:REAL;
	K:REAL;
END_VAR
CalcRRGSPwithCoeff:=V*K;
END_METHOD

END_FUNCTION_BLOCK

// Function Blocks/GeneralBuffer/fbGeneralBuffer
(*
fbGeneralBuffer предназначен для работы с байтовым буффером
*)
FUNCTION_BLOCK fbGeneralBuffer
VAR_INPUT
	pBuffer:	POINTER TO BYTE;
	pBufferLength: INT;
END_VAR
VAR_OUTPUT
	xEmpty: BOOL;
	xInit:BOOL;
END_VAR
VAR
	Init:BOOL:=FALSE;
	Buffer: udtGeneralBuffer;
END_VAR

IF pBuffer = 0 OR pBufferLength =0 THEN
	xEmpty:=TRUE;
	RETURN;
ELSE
	xEmpty:=FALSE;
END_IF
IF NOT Init AND NOT xEmpty THEN
	Buffer.Buffer:=pBuffer;
	Buffer.MaxLength:=pBufferLength;
	Buffer.Offset:=0;
	Init:=TRUE;
	xInit:=true;
END_IF

METHOD PUBLIC AddElement : INT
VAR_INPUT
	pData:	BYTE;

END_VAR
IF THIS^.Buffer.Offset > THIS^.Buffer.MaxLength THEN
	AddElement:=-1;
	RETURN;
END_IF
MEMUtils.MemCpy(pbyDest:=THIS^.Buffer.Buffer+THIS^.Buffer.Offset,
				pbySrc:=ADR(pData),
				dwSize:=1);
THIS^.Buffer.Offset :=	THIS^.Buffer.Offset+1;
AddElement:=100;
END_METHOD

METHOD PUBLIC AddStruct : INT
VAR_INPUT
	pData:	POINTER TO BYTE;
	Length: INT;
END_VAR
IF THIS^.Buffer.Offset+Length > THIS^.Buffer.MaxLength THEN
	AddStruct:=-1;
	RETURN;
END_IF
MEMUtils.MemCpy(pbyDest:=THIS^.Buffer.Buffer+THIS^.Buffer.Offset,
				pbySrc:=pData,
				dwSize:=Length);
THIS^.Buffer.Offset :=	THIS^.Buffer.Offset+Length;
AddStruct:=100;
END_METHOD

METHOD PUBLIC ClearBuffer : INT
VAR_INPUT
END_VAR

MEMUtils.MemSet(pbyBuffer:=THIS^.Buffer.Buffer,
				byValue:=0,
				dwSize:=THIS^.Buffer.MaxLength);
THIS^.Buffer.Offset:=0;
ClearBuffer:=200;
END_METHOD

PROPERTY PUBLIC getBufferAddres : DINT
GET
getBufferAddres:=THIS^.Buffer.Buffer;
END_GET
END_PROPERTY

PROPERTY PUBLIC getBufferLength : DINT
GET
getBufferLength:=THIS^.Buffer.Offset;
END_GET
END_PROPERTY

END_FUNCTION_BLOCK

// Function Blocks/Gorn/Gorn
FUNCTION_BLOCK Gorn
VAR_INPUT
	refGorn: 				REFERENCE TO udtGorn;
	refGornSetting:			REFERENCE TO udtGornSetting;
	xPowerOnFeedback: 		BOOL;						//Включение контактора
	xInterlock:		 		BOOL;
	xModbusConnected:		BOOL;
	refGornRegisters: 		REFERENCE TO udtGornModbus;
	
END_VAR
VAR_OUTPUT
	xInternalError:				BOOL;// OUTPUT: Внутренняя ошибка
	xStabVoltageError:			BOOL;// OUTPUT: Ошибка стабилизации напряжения
	xStabCurrentError:			BOOL;// OUTPUT:	Ошибка стабилизации силы тока
	xPowerError:				BOOL;// OUTPUT: Ошибка силовой части
	xHeatProtect:				BOOL;// OUTPUT: Тепловая защита
	xRemoteStatus:				BOOL;// OUTPUT: Статус удаленной работы
	xError:						BOOL;// OUTPUT: Ошибка

END_VAR
VAR
	xCommand:				BOOL;
	SpCurrent:				INT;
	SpVoltage:				INT;
END_VAR

